METHOD M_Execute
//////////////////
//  Method Calls 
/////////////////

VAR 
	// Method local variables (reinitialized at each cycle) 

END_VAR
IF NOT bInit THEN
	M_Init();
END_IF


SUPER^.M_Execute() ;
END_METHOD

METHOD M_Init
VAR_INPUT
END_VAR

VAR

END_VAR
ParamPnom := 2200.0 ;
IN_SetptPlimit_Local :=  2200.0;
ParamQnom := 1650;
bInit := TRUE;
END_METHOD

{attribute 'object_name' := 'M_Read'}
METHOD M_Read
//////////
// Read Method for SMA : Modbus reading
//////////
VAR
	// Method local variables (reinitialized at each cycle) 
	MW 					: FB_MergeWordsToDint; 
	
	
	KK					: BYTE;						 // Index to loop over modbus blocks. 	
	JJ					: BYTE;						// Index loop over Number of SB
	CalOpTm: INT;
	
	AX_Qty				: ARRAY[1..2] OF WORD := [100, 		6 		];
	AX_Addr				: ARRAY[1..2] OF WORD := [57, 	40112 	];
	AX_UnitId			: ARRAY[1..2] OF BYTE := [1, 		1		];

	
	mesH: REAL;
	test: LREAL;
	test1: UINT;
END_VAR

IF MesDataExd.MesData.MesCP_Read THEN 
	
	FOR KK := 1 TO 1 DO
		ModbusReadRegs[KK]
		(
			nTcpPort := ParamTcpPort,
			pDestAddr := ADR(MesBlock_Temp[KK]),
			cbLength := SIZEOF(MesBlock_Temp[KK]),
			sIPAddr := ParamIPAddress,
			tTimeout := ParamTimeout,
			nQuantity := AX_Qty[KK],
			nMBAddr := AX_Addr[KK],
			nUnitID := AX_UnitID[KK],
			ClockRead := ClockRead,
			ErrorId => ModbusAlarmsID[KK],
			ModbusReadAlarm => ModbusAlarm[KK]
		);
	END_FOR
	
	MW(WORD_STRONG := MesBlock_Temp[1][1 ] 										, SIZE :=  1, FIX :=  1, SIGNED := TRUE, 	SmaDevice := TRUE, VAR_OUT := MesDataExd.MesData.MesSetptP);
	MW(WORD_STRONG := MesBlock_Temp[1][2 ] 										, SIZE :=  1, FIX :=  1, SIGNED := TRUE, 	SmaDevice := TRUE, VAR_OUT := MesDataExd.MesData.MesP);
	MW(WORD_STRONG := MesBlock_Temp[1][4 ] 										, SIZE :=  1, FIX :=  1, SIGNED := TRUE, 	SmaDevice := TRUE, VAR_OUT := MesDataExd.MesData.MesSetptQ);
	MW(WORD_STRONG := MesBlock_Temp[1][5 ] 										, SIZE :=  1, FIX :=  1, SIGNED := TRUE, 	SmaDevice := TRUE, VAR_OUT := MesDataExd.MesData.MesQ);
	MW(WORD_STRONG := MesBlock_Temp[1][10] 										, SIZE :=  1, FIX :=  1, SIGNED := TRUE, 	SmaDevice := TRUE, VAR_OUT := MesDataExd.MesData.MesNbInvAvail);
	MW(WORD_STRONG := MesBlock_Temp[1][16] 										, SIZE :=  1, FIX :=  0, SIGNED := FALSE, 	SmaDevice := TRUE, VAR_OUT := MesDataExd.MesData.MesPState);
	MW(WORD_STRONG := MesBlock_Temp[1][18] 										, SIZE :=  1, FIX :=  0, SIGNED := FALSE, 	SmaDevice := TRUE, VAR_OUT := MesDataExd.MesData.MesQState);
	MW(WORD_STRONG := MesBlock_Temp[1][20] 										, SIZE :=  1, FIX :=  0, SIGNED := FALSE, 	SmaDevice := TRUE, VAR_OUT := MesDataExd.MesData.MesGeneState);
	MW(WORD_STRONG := MesBlock_Temp[1][30], WORD_WEAK := MesBlock_Temp[1][31]	, SIZE :=  2, FIX :=  0, SIGNED := TRUE, 	SmaDevice := TRUE, VAR_OUT := MesDataExd.MesData.MesPNomControlled);
	MW(WORD_STRONG := MesBlock_Temp[1][32], WORD_WEAK := MesBlock_Temp[1][33]	, SIZE :=  2, FIX :=  0, SIGNED := TRUE, 	SmaDevice := TRUE, VAR_OUT := MesDataExd.MesData.MesPControlled);
	MW(WORD_STRONG := MesBlock_Temp[1][34], WORD_WEAK := MesBlock_Temp[1][35]	, SIZE :=  2, FIX :=  0, SIGNED := TRUE, 	SmaDevice := TRUE, VAR_OUT := MesDataExd.MesData.MesQControlled);
	MW(WORD_STRONG := MesBlock_Temp[1][40], WORD_WEAK := MesBlock_Temp[1][41]	, SIZE :=  2, FIX :=  0, SIGNED := TRUE, 	SmaDevice := TRUE, VAR_OUT := MesDataExd.MesData.MesQNomControlled);
	MW(WORD_STRONG := MesBlock_Temp[1][42] 										, SIZE :=  1, FIX :=  0, SIGNED := FALSE, 	SmaDevice := TRUE, VAR_OUT := MesDataExd.MesData.MesWatchdog);

	
END_IF
END_METHOD

METHOD M_StartStop
//////////////////
// Start and Stop AMG
/////////////////
VAR 
	// Method local variables (reinitialized at each cycle) 

END_VAR
// Set SetptLimit to zero if Stop command
SUPER^.M_StartStop() ; 
//RS_StartStop(SET:=CmdStart,Reset1:=CmdStop); IN BASE
END_METHOD

METHOD M_StateManager
//////////////////
// Detect which is the state of the inverter. IF loss of communication MesState =0 , the last inverter state is kept .  
/////////////////

VAR 
	// Method local variables (reinitialized at each cycle) 

	
	MesGeneState: WORD;

END_VAR
MesState 			:= 0  ; 

MesGeneState:= REAL_TO_WORD(MesDataExd.MesGeneState);


IF MesGeneState.0 THEN
	MesState.5 := TRUE;
ELSIF MesGeneState.1 THEN
	MesState.5 := FALSE;
END_IF

IF MesGeneState.8 = 1 THEN
	MesState.3 := TRUE;
ELSIF MesGeneState.9 THEN
	MesState.3 := FALSE;
END_IF

IF MesDataExd.MesPState = 2 THEN 
	MesState.1 := TRUE;
ELSE 
	MesState.1 := FALSE;
END_IF
IF MesDataExd.MesQState = 2 THEN 
	MesState.2 := TRUE;
ELSE 
	MesState.2 := FALSE;
END_IF
SUPER^.M_StateManager() ;
END_METHOD

{attribute 'object_name' := 'M_Write'}
METHOD M_Write
//////////////////
// Write Curtail Command through modbus to PV inverters.  
//////////////////
VAR 
	// Method local variables (reinitialized at each cycle) 

	SFW : FB_SplitRealToWords_IEEE754;

	dwordTest: DWORD;
	wordTest1: WORD;
	WordTest2: WORD;
END_VAR


AX_CmdWrite[1] := 0;
SFW(IN_Real := A1_SUBMV.A1_GRID.MesDataExd.MesData.OUT_SetptP , 	OUT_WordStrong =>AX_CmdWrite[3], 	OUT_WordWeak =>AX_CmdWrite[2]);

AX_CmdWrite[14] := 0;
SFW(IN_Real := A1_SUBMV.A1_GRID.MesDataExd.MesData.OUT_SetptQ, 	OUT_WordStrong =>AX_CmdWrite[16], 	OUT_WordWeak =>AX_CmdWrite[15]);

(*
AX_CmdWrite[31] := REAL_TO_WORD(RtuData.SetptQfU_Acknw*100);
AX_CmdWrite[37] := UINT_TO_WORD(REAL_TO_UINT(RtuData.SetptPF_Acknw*10000));
AX_CmdWrite[49] := REAL_TO_WORD(2.0); 								// Configuration of active power control (Active power control with P(f) generic 2-5)
AX_CmdWrite[50] := UINT_TO_WORD(RtuData.OUT_TypeConsigneReactive); //Type de consigne  en cours 0: Aucune, 1: Q, 2: QfU, 3: PF

*)
//
//
SFW(IN_Real := A1_SUBMV.MesDataExd.MesData.MesPsol, 			OUT_WordStrong =>AX_CmdWrite1[2], 	OUT_WordWeak =>AX_CmdWrite1[1]);


SFW(IN_Real := A1_SUBMV.MesDataExd.MesData.MesQsol, 			OUT_WordStrong =>AX_CmdWrite1[4], 	OUT_WordWeak =>AX_CmdWrite1[3]);
AX_CmdWrite1[5] := REAL_TO_WORD(REAL_TO_UINT(A1_SUBMV.MesDataExd.MesData.MesU*100));
AX_CmdWrite1[6] := REAL_TO_WORD(REAL_TO_UINT(A1_SUBMV.MesDataExd.MesData.MesFreq*100)); 
//AX_CmdWrite1[7] := REAL_TO_WORD(REAL_TO_UINT(A1_SUBMV.MesDataExd.MesData.MesTanPhi*1000)); 	// Csophi 

ModbusWrite[1]
(
	pSrcAddr := ADR(AX_CmdWrite),
	sIPAddr := ParamIPAddress,
	nTCPport := ParamTcpPort,
	tTimeout := ParamTimeout,
	nMBAddr := 133,
	cbLength := SIZEOF(AX_CmdWrite),
	nQuantity :=  50,
	WriteCmd := ClockWrite,
	nUnitID := 1
);

ModbusWrite[2]
(
	pSrcAddr := ADR(AX_CmdWrite1),
	sIPAddr := ParamIPAddress,
	nTCPport := ParamTcpPort,
	tTimeout := ParamTimeout,
	nMBAddr := 189,
	cbLength := SIZEOF(AX_CmdWrite1),
	nQuantity :=  7,
	WriteCmd := ClockWrite,
	nUnitID := 1
);

SUPER^.M_Write() ;
END_METHOD

END_FUNCTION_BLOCK

// ---- 01_Equipement_Library/ProtectRelay/FB_ProtectRelay_DM2.TcPOU
FUNCTION_BLOCK FB_ProtectRelay_DM2 EXTENDS FB_ProtectRelay_Base
//////////////////
// REF615 + REU615 : communication not allowed by EDF 

VAR_OUTPUT
	//Child objects

END_VAR

VAR_INPUT
	IN_AlarmIMax_IO								: BOOL; //Max I Alarm, Losing autorisation and not possible to consumed
	IN_AlarmUmin_IO									: BOOL; //Min U , Keeping autorisation, If we have 3 gte in 30 min ==> Stop fedding and consumed during 2h
	IN_MesWatchdogREU615_IO						: BOOL:=TRUE ;// Watchdog . 0= alarm
	MesDataExd		: ProtectRelay_Standard ; 	
END_VAR

VAR
	//M_ALARMMANAGEMENT VARIABLES//

	
	// EVALUATE //
	TON_GteIsLong	: TON ; 
	
	


		
END_VAR

METHOD M_AlarmManagement
//////////////////
// Manages Sepam Alarms. Alarms opens HT CB until Sepam manual Reset . Warning Opens CB-L but does not maintain warning
/////////////////

VAR 
	// Method local variables (reinitialized at each cycle) 
	FB_AlarmCodeManager 	: FB_AlarmCodeManager ; 

 
END_VAR


// ALARM CODE //
	FB_AlarmCodeManager(
		bAlarm1				:= MesDataExd.MesData.MesAlarmImax , 						// Max I>>0  fault 	 	
		bAlarm2				:= MesDataExd.MesData.MesAlarmUmin ,							// GTE fault 
		bAlarm3				:= MesDataExd.MesData.MesAlarmCom,						// Communication Alarm #COM
		bAlarm4				:= NOT IN_MesWatchDog_IO, 						// Watchdog REF615 not received      #COM 
		bAlarm5				:= NOT IN_MesWatchdogREU615_IO, 				// Watchdog REU615 not received	 #COM
		bAlarm6				:= FALSE, 									// 
		bAlarm7				:= FALSE, 									//
		bAlarm8				:= FALSE,                                   //
		bAlarm9				:= FALSE,                                   //
		bAlarm10			:= FALSE,                                   //
		bAlarm11			:= FALSE,                                   //
		bAlarm12			:= FALSE,                                   //
		bAlarm13			:= FALSE, 									//
		bAlarm14			:= FALSE, 									//
		bAlarm15			:= FALSE ,									// 
		wAlarmCode			=>MesDataExd.MesData.MesAlarmCode);

// WARNING CODE //
	FB_AlarmCodeManager(
		bAlarm1			:= FALSE , //
		bAlarm2			:= FALSE , //	
		bAlarm4			:= MesDataExd.MesData.MesAlarmUmin_Long, 						// GTE long 
		bAlarm5			:= FALSE, 									//
		bAlarm6			:= FALSE,                                   //
		bAlarm7			:= FALSE,                                   //
		bAlarm8			:= FALSE,                                   //
		bAlarm9			:= FALSE,                                   //
		bAlarm10		:= FALSE,                                   //
		bAlarm11		:= FALSE,                                   //
		bAlarm12		:= FALSE,                                   //
		bAlarm13		:= FALSE,                                   //
		bAlarm14		:= FALSE,                                   //
		bAlarm15		:= FALSE, 									//
		wAlarmCode		=>MesDataExd.MesData.MesWarningCode);

// EVENT CODE //
	FB_AlarmCodeManager(
		bAlarm1			:=FALSE, 		//  
		bAlarm2			:=FALSE, 		//  
		bAlarm3			:=FALSE, 		//  
		bAlarm4			:=FALSE, 		// 
		bAlarm5			:=FALSE,        //
		bAlarm6			:=FALSE,        //
		bAlarm7			:=FALSE,        //
		bAlarm8			:=FALSE,        //
		bAlarm9			:=FALSE,        //
		bAlarm10		:=FALSE,        //
		bAlarm11		:=FALSE,        //
		bAlarm12		:=FALSE,        //
		bAlarm13		:=FALSE,        //
		bAlarm14		:=FALSE,        //
		bAlarm15		:=FALSE, 
		wAlarmCode		=>MesDataExd.MesData.MesEventCode);
END_METHOD

METHOD M_CP
//////////////////
//  Emulator
/////////////////

VAR 
	// Method local variables (reinitialized at each cycle) 
	
END_VAR


SUPER^.M_CP() ; 




Trig_Cmd_Read(CLK:=IN_CmdToggleRead);
Trig_Cmd_Write(CLK:=IN_CmdToggleWrite);
	
IF Trig_Cmd_Read.Q THEN
	IN_CmdToggleRead := FALSE;
	MesDataExd.MesData.MesCP_Read := NOT MesDataExd.MesData.MesCP_Read;
END_IF


IF Trig_Cmd_Write.Q THEN
	IN_CmdToggleWrite := FALSE;
	MesDataExd.MesData.MesCP_Write := NOT MesDataExd.MesData.MesCP_Write;
END_IF
END_METHOD

METHOD M_Evaluate
VAR_INPUT
END_VAR
//Need to check the GTE FAULT


// GTE IS LONG AFTER 50S
TON_GteIsLong(IN:=IN_AlarmUmin_IO ,PT:=T#50S); 
MesDataExd.MesData.MesAlarmUmin_Long := TON_GteIsLong.Q ; 


//Update MesData

MesDataExd.MesData.MesAlarmUmin 			:= IN_AlarmUmin_IO;

TON_ComAlarm(IN:=NOT IN_MesWatchDog_IO OR NOT IN_MesWatchdogREU615_IO , PT:=ParamTempoComAlarm ) ; 
MesDataExd.MesData.MesAlarmCom		:=TON_ComAlarm.Q  ; 
MesDataExd.MesData.MesAlarmImax		:= IN_AlarmIMax_IO;
END_METHOD

END_FUNCTION_BLOCK

// ---- 01_Equipement_Library/ProtectRelay/FB_ProtectRelay_Base.TcPOU
FUNCTION_BLOCK FB_ProtectRelay_Base
//////////////////
// SEPAM system for High Voltage or Low Voltage Grid Protection. 
//////////////////
VAR_INPUT PERSISTENT
	// Parameters of the Object (instance/model specific) 
		ParamTempoComAlarm					: TIME := T#10S;	(* (s) Config : Tempo to detect LOC Alarm*)
		ParamTimeOut						: TIME := T#5S;		(* (s) Modbus Timeout*)
		ParamClockReadTime					: TIME := T#2S;		(* (s) Modbus Read Frequency*)
		ParamClockWriteTime					: TIME := T#1S;		(* (s) Modbus Write Frequency*)
				   		                    		
END_VAR                                                        

VAR_OUTPUT
	//Child objects
	
END_VAR

VAR_INPUT
	IN_CmdReset_L							: BOOL;				// (NA) External Reset Command	
    IN_CmdToggleRead						: BOOL;
    IN_CmdToggleWrite						: BOOL;
	                                    
	// I/O Inputs                       
		// GTE Protection LV            
		// WatchDog                     
	IN_MesWatchDog_IO						: BOOL :=TRUE;		// Watchdog is at True := Sepam OK
END_VAR

VAR
	//M_ALARMMANAGEMENT VARIABLES//                                                  
		TON_ComAlarm						: TON ; 			// Tempo before detecting loss of communication. 
	
	//M_READ //
		TP1									: TP;
		TP2									: TP;
		ClockRead				AT %Q*		: BOOL;
		ClockWrite							: BOOL;
	///MesDataExd						: ProtectRelay;		

    //M_CP VARIABLES//
		Trig_Cmd_Read						: R_TRIG;                                                                                        
		Trig_Cmd_Write						: R_TRIG;                                                                                        
	//M_INIT VARIABLES // 	        		
		bInit								: BOOL := TRUE ; 		// (NA) Initialize object parameters at first cycle 
END_VAR

METHOD M_AlarmManagement
//////////////////
// Manages Sepam Alarms. Alarms opens HT CB until Sepam manual Reset . Warning Opens CB-L but does not maintain warning
/////////////////

VAR 
	// Method local variables (reinitialized at each cycle) 
	FB_AlarmCodeManager 	: FB_AlarmCodeManager ; 

 
END_VAR
END_METHOD

METHOD M_CP 
VAR_INPUT
END_VAR
END_METHOD

METHOD M_Evaluate
VAR_INPUT
END_VAR
END_METHOD

METHOD M_Execute
//////////////////
//  Method Calls 
/////////////////

VAR 
	// Method local variables (reinitialized at each cycle) 

END_VAR
	TP1(IN:=NOT TP1.Q , PT:= ParamClockReadTime);
	ClockRead 		:= TP1.Q;
	TP2(IN:=NOT TP2.Q , PT:= ParamClockWriteTime);
	ClockWrite		:= TP2.Q;

// INITIALIZE // 
	IF bInit THEN
		M_Init() ; 
		bInit		:= FALSE ; 
		
	ELSIF CmdInit_G OR IN_CmdReset_L THEN 
		bInit		:= TRUE ;
		
	END_IF

// METHODS CALLS // 
	M_CP();
	M_Read(); 
	
	M_Evaluate(); 
	M_Write();
	
	M_AlarmManagement();
END_METHOD

METHOD M_Init
VAR_INPUT
END_VAR
END_METHOD

METHOD M_Read
//////////////////
//  Method Calls 
/////////////////

VAR 
	// Method local variables (reinitialized at each cycle) 

END_VAR
END_METHOD

METHOD M_Write 
VAR_INPUT
END_VAR
END_METHOD

END_FUNCTION_BLOCK

// ---- 01_Equipement_Library/ProtectRelay/FB_ProtectRelay_Flair23DM.TcPOU
FUNCTION_BLOCK FB_ProtectRelay_Flair23DM EXTENDS FB_ProtectRelay_Base
//////////////////
// SEPAM system for High Voltage or Low Voltage Grid Protection. 
//////////////////
VAR_INPUT PERSISTENT
	ParamTcpPort				: UINT:=502;                       (* (NA) Tcp port *)
	ParamIPAddress				: STRING; 						   (* (NA) IP address*)
	ParamUnitID					: BYTE; 						   (* (NA) Unit ID*)
END_VAR

VAR_INPUT 
	MesDataExd	AT %Q*	: ProtectRelay_Flair23DM;     		//  MesDataExd.MesData.xd
	
END_VAR

VAR_OUTPUT
	
END_VAR

VAR_INPUT

END_VAR

VAR

	FB_ModbusRead	          	: ARRAY[1..3] OF FB_ModbusRead; 	// Modbus Read
									
	CalCP_Read					: BOOL;								
	CalCP_Write					: BOOL;
	
	MesBlock1_Temp 				: ARRAY [1..1] OF WORD ; 
	MesBlock2_Temp 				: ARRAY [1..15] OF WORD; 
	MesBlock3_Temp 				: ARRAY [1..2] OF WORD ; 
	
	AX_ModbusReadAlarm			: ARRAY[1..3] OF BOOL  ;
	AX_ModbusReadAlarmId		: ARRAY[1..3] OF UDINT ;	
END_VAR

METHOD M_AlarmManagement
//////////////////
// Manages Sepam Alarms. Alarms opens HT CB until Sepam manual Reset. Warning Opens CB-L but does not maintain warning.
/////////////////

VAR 
	// Method local variables (reinitialized at each cycle) 
	FB_AlarmCodeManager 	: FB_AlarmCodeManager ; 
 	ComWarning				: BOOL;
	ComAlarms				: BOOL;
END_VAR
// ALARM CODE //
	FB_AlarmCodeManager(
		bAlarm1			:= NOT MesDataExd.MesData.MesAlarmCom,	// Com error: the device did not respond successfully to most recent read/write request
		bAlarm2			:= FALSE,						//				
		bAlarm3			:= FALSE,   					//
		bAlarm4			:= FALSE,   					//
		bAlarm5			:= FALSE,   					//
		bAlarm6			:= FALSE, 						//
		bAlarm7			:= FALSE,   					//
		bAlarm8			:= FALSE,   					//
		bAlarm9			:= FALSE,   					//
		bAlarm10		:= FALSE,   					//
		bAlarm11		:= FALSE,   					//
		bAlarm12		:= FALSE,   					//
		bAlarm13		:= FALSE,   					//
		bAlarm14		:= FALSE,   					//
		bAlarm15		:= FALSE, 						//
		wAlarmCode		=>MesDataExd.MesData.MesAlarmCode);   	//

// WARNING CODE //
	FB_AlarmCodeManager(
		bAlarm1			:= FALSE,						//
		bAlarm2			:= FALSE,   					//
		bAlarm4			:= FALSE,   					//
		bAlarm5			:= FALSE,   					//
		bAlarm6			:= FALSE, 						//
		bAlarm7			:= FALSE,   					// 
		bAlarm8			:= FALSE,   					// 
		bAlarm9			:= FALSE,   					// 
		bAlarm10		:= FALSE,   					// 
		bAlarm11		:= FALSE,   					// 
		bAlarm12		:= FALSE,   					// 
		bAlarm13		:= FALSE,   					// 
		bAlarm14		:= FALSE,   					// 
		bAlarm15		:= FALSE, 						// 
		wAlarmCode		=>MesDataExd.MesData.MesWarningCode);	    //

// EVENT CODE //
	FB_AlarmCodeManager(
		bAlarm1			:=FALSE,						// 		
		bAlarm2			:=FALSE,   						// 		
		bAlarm3			:=FALSE,   						// 		
		bAlarm4			:=FALSE,   						// 		
		bAlarm5			:=FALSE, 						// 
		bAlarm6			:=FALSE,   						// 
		bAlarm7			:=FALSE,   						// 
		bAlarm8			:=FALSE,   						// 
		bAlarm9			:=FALSE,   						// 
		bAlarm10		:=FALSE,   						// 
		bAlarm11		:=FALSE,   						// 
		bAlarm12		:=FALSE,   						// 
		bAlarm13		:=FALSE,   						// 
		bAlarm14		:=FALSE, 						// 
		bAlarm15		:=FALSE, 						//		
		wAlarmCode		=>MesDataExd.MesData.MesEventCode); 		//
END_METHOD

METHOD M_CP
//////////////////
//  Emulator
/////////////////

VAR 
	// Method local variables (reinitialized at each cycle) 
	
END_VAR


SUPER^.M_CP() ; 




Trig_Cmd_Read(CLK:=IN_CmdToggleRead);
Trig_Cmd_Write(CLK:=IN_CmdToggleWrite);
	
IF Trig_Cmd_Read.Q THEN
	IN_CmdToggleRead := FALSE;
	MesDataExd.MesData.MesCP_Read := NOT MesDataExd.MesData.MesCP_Read;
END_IF


IF Trig_Cmd_Write.Q THEN
	IN_CmdToggleWrite := FALSE;
	MesDataExd.MesData.MesCP_Write := NOT MesDataExd.MesData.MesCP_Write;
END_IF
END_METHOD

METHOD M_Evaluate
VAR_INPUT
END_VAR

VAR
END_VAR

SUPER^.M_Evaluate() ;
END_METHOD

METHOD M_Execute
//////////////////
//  Method Calls 
/////////////////

VAR 
	// Method local variables (reinitialized at each cycle) 

END_VAR
IF NOT bInit THEN
	M_Init();
END_IF


SUPER^.M_Execute() ;
END_METHOD

METHOD M_Init
VAR_INPUT
END_VAR
binit := true;
END_METHOD

METHOD M_Read
//////////////////
//  Method Calls 
/////////////////

VAR_INPUT
	
END_VAR
VAR 
	MW					: FB_MergeWordsToFloat;
END_VAR

// CP-Read / Write 



// System BMS 
IF MesDataExd.MesData.MesCP_Read  THEN	

	
	FB_ModbusRead[1]
		(
			nTCPPort		:= ParamTcpPort,
			ClockRead		:= MesDataExd.MesData.MesCP_Read AND ClockRead, 
			Reset			:= CmdClearFault_G OR IN_CmdReset_L,
			sIPAddr			:= ParamIPAddress,
			nUnitID			:= ParamUnitID, 
			tTimeout		:= T#5S,
			nQuantity		:= 1, 
			nMBAddr			:= 41000 , 
			cbLength		:= SIZEOF(MesBlock1_Temp), 
			pDestAddr		:= ADR(MesBlock1_Temp) , 
			ModbusReadAlarm	=> AX_ModbusReadAlarm[1] , 
			ErrorId			=> AX_ModbusReadAlarmId[1]
		);
		
	FB_ModbusRead[2]
		(
			nTCPPort		:= ParamTcpPort,
			ClockRead		:= MesDataExd.MesData.MesCP_Read AND ClockRead, 
			Reset			:= CmdClearFault_G OR IN_CmdReset_L,
			sIPAddr			:= ParamIPAddress,
			nUnitID			:= ParamUnitID, 
			tTimeout		:= T#5S,
			nQuantity		:= 14, 
			nMBAddr			:= 41200, 
			cbLength		:= SIZEOF(MesBlock2_Temp), 
			pDestAddr		:= ADR(MesBlock2_Temp) , 
			ModbusReadAlarm	=> AX_ModbusReadAlarm[2], 
			ErrorId			=> AX_ModbusReadAlarmId[2]
		);
	
	FB_ModbusRead[3]
		(
			nTCPPort		:= ParamTcpPort,
			ClockRead		:= MesDataExd.MesData.MesCP_Read AND ClockRead, 
			Reset			:= CmdClearFault_G OR IN_CmdReset_L,
			sIPAddr			:= ParamIPAddress ,
			nUnitID			:= ParamUnitID, 
			tTimeout		:= T#5S,
			nQuantity		:= 2, 
			nMBAddr			:= 41350 , 
			cbLength		:= SIZEOF(MesBlock3_Temp), 
			pDestAddr		:= ADR(MesBlock3_Temp) , 
			ModbusReadAlarm	=> AX_ModbusReadAlarm[3], 
			ErrorId			=> AX_ModbusReadAlarmId[3]
		);
			
	//COM
	MesDataExd.MesStateCom 			:= WORD_TO_BOOL(MesBlock1_Temp[1]);
	//I
	MesDataExd.MesData.MesI1 		:= WORD_TO_INT(Mesblock2_Temp[1]) ;
	MesDataExd.MesData.MesI2 	    := WORD_TO_INT(Mesblock2_Temp[2]) ;
	MesDataExd.MesData.MesI3       := WORD_TO_INT(Mesblock2_Temp[3]) ;
	MesDataExd.MesData.MesI0 	    := WORD_TO_INT(Mesblock2_Temp[4]) ;
	//Imax
	MesDataExd.MesData.MesImax1 	:= WORD_TO_INT(Mesblock2_Temp[5]) ;	
	MesDataExd.MesData.MesImax2 	:= WORD_TO_INT(Mesblock2_Temp[6]) ;	
	MesDataExd.MesData.MesImax3 	:= WORD_TO_INT(Mesblock2_Temp[7]) ;	
	//V
	MesDataExd.MesV1				:= WORD_TO_REAL(Mesblock2_Temp[8]) * 0.01 ;	
	MesDataExd.MesV2				:= WORD_TO_REAL(Mesblock2_Temp[9]) * 0.01 ;
	MesDataExd.MesV3				:= WORD_TO_REAL(Mesblock2_Temp[10])* 0.01 ;
	MesDataExd.MesV0				:= WORD_TO_REAL(Mesblock2_Temp[11])* 0.01 ;
		
	MesDataExd.MesData.MesU12		:= WORD_TO_REAL(Mesblock2_Temp[12])* 0.01 ;					// U21 
	MesDataExd.MesData.MesU23		:= WORD_TO_REAL(Mesblock2_Temp[13])* 0.01 ; 				// U32 
	MesDataExd.MesData.MesU31		:= WORD_TO_REAL(Mesblock2_Temp[14])* 0.01 ; 				// U31  
		
	MesDataExd.ControlWord 			:= MesBlock3_Temp[1];
	MesDataExd.StatusWord 			:= MesBlock3_Temp[2];
		
END_IF
END_METHOD

END_FUNCTION_BLOCK

// ---- 01_Equipement_Library/ProtectRelay/FB_ProtectRelay_MaxI.TcPOU
FUNCTION_BLOCK FB_ProtectRelay_MaxI EXTENDS FB_ProtectRelay_Base
//////////////////
// SEPAM system for High Voltage or Low Voltage Grid Protection . 
//////////////////


VAR_INPUT PERSISTENT 
	ParamTcpPort				: UINT:=502;	(* TCP Port parameter*)
	ParamIPAddress				: STRING; 		(* IP Address*)
	ParamUnitID					: BYTE; 		(* Unit ID*)
	
END_VAR

VAR_INPUT
	MesDataExd					: ProtectRelay_Standard;
END_VAR

VAR
	ClockReadInput				: BOOL;
	AX_MbRead					: ARRAY[1..1] OF FB_ModbusRead;
	AX_Word						: ARRAY[1..1] OF ARRAY[1..120] OF WORD;
	AX_ADDR						: ARRAY[1..1] OF UINT := [300];
	AX_QTY						: ARRAY[1..1] OF UINT := [16];	
	AX_UnId						: ARRAY[1..1] OF BYTE := [3];
END_VAR

METHOD M_AlarmManagement
//////////////////
// Manages Sepam Alarms. Alarms opens HT CB until Sepam manual Reset . Warning Opens CB-L but does not maintain warning
/////////////////

VAR 
	// Method local variables (reinitialized at each cycle) 
	FB_AlarmCodeManager 	: FB_AlarmCodeManager ; 
	RS_Trip					: SR;
END_VAR

MesDataExd.MesData.MesComAlarm		:= AX_MbRead[1].ModbusReadAlarm  ;

// ALARM CODE //
	FB_AlarmCodeManager(
		bAlarm1				:= MesDataExd.MesData.MesComAlarm,		// Communication alarm
		bAlarm2				:= FALSE,
		bAlarm3				:= FALSE,
		bAlarm4				:= FALSE,
		bAlarm5				:= FALSE,         					
		bAlarm6				:= FALSE, 							
		bAlarm7				:= FALSE, 
		bAlarm8				:= FALSE, 
		bAlarm9				:= FALSE, 
		bAlarm10			:= FALSE, 
		bAlarm11			:= FALSE, 
		bAlarm12			:= FALSE, 
		bAlarm13			:= FALSE, 
		bAlarm14			:= FALSE, 
		bAlarm15			:= FALSE , 	
		wAlarmCode			=> MesDataExd.MesData.MesAlarmCode);
END_METHOD

METHOD M_CP
//////////////////
//  Emulator
/////////////////

VAR 
	// Method local variables (reinitialized at each cycle) 
	
END_VAR


SUPER^.M_CP() ; 




Trig_Cmd_Read(CLK:=IN_CmdToggleRead);
Trig_Cmd_Write(CLK:=IN_CmdToggleWrite);
	
IF Trig_Cmd_Read.Q THEN
	IN_CmdToggleRead := FALSE;
	MesDataExd.MesData.MesCP_Read := NOT MesDataExd.MesData.MesCP_Read;
END_IF


IF Trig_Cmd_Write.Q THEN
	IN_CmdToggleWrite := FALSE;
	MesDataExd.MesData.MesCP_Write := NOT MesDataExd.MesData.MesCP_Write;
END_IF
END_METHOD

METHOD M_Evaluate
VAR_INPUT
END_VAR

VAR
END_VAR
END_METHOD

METHOD M_Init
VAR_INPUT
END_VAR
END_METHOD

METHOD M_Read
//////////////////
//  Method Calls 
/////////////////

VAR_INPUT
	
END_VAR
VAR 
	MW					: FB_MergeWordsToFloat;
	


	KK: INT;
END_VAR
IF MesDataExd.MesData.MesCP_Read THEN

	FOR KK := 1 TO 1 DO
		AX_MbRead[KK]
		(
			pDestAddr := ADR(AX_Word[KK]),
			sIPAddr := ParamIPAddress,
			tTimeout := T#2S,
			nTcpPort := ParamTcpPort,
			nQuantity := AX_QTY[KK],
			nMBAddr := AX_ADDR[KK],
			cbLength := SIZEOF(AX_Word[KK]),
			nUnitID := AX_UnId[KK],
			ClockRead := ClockRead
		);
	END_FOR
	
	MW(WORD_STRONG_F := AX_WORD[1][1], WORD_WEAK_F := AX_Word[1][2], NUMBER_F := MesDataExd.MesData.MesI1);
	MW(WORD_STRONG_F := AX_WORD[1][3], WORD_WEAK_F := AX_Word[1][4], NUMBER_F := MesDataExd.MesData.MesI2);
	MW(WORD_STRONG_F := AX_WORD[1][5], WORD_WEAK_F := AX_Word[1][6], NUMBER_F := MesDataExd.MesData.MesI3);
	MW(WORD_STRONG_F := AX_WORD[1][7], WORD_WEAK_F := AX_Word[1][8], NUMBER_F := MesDataExd.MesData.MesI0);
	
END_IF

MesDataExd.MesData.MesI := (MesDataExd.MesData.MesI1 + MesDataExd.MesData.MesI2 + MesDataExd.MesData.MesI3)/3;
END_METHOD

END_FUNCTION_BLOCK

// ---- 01_Equipement_Library/ProtectRelay/FB_ProtectRelay_Micom.TcPOU
FUNCTION_BLOCK FB_ProtectRelay_Micom EXTENDS FB_ProtectRelay_Base
//////////////////
// SEPAM system for High Voltage or Low Voltage Grid Protection. 
//////////////////

VAR_INPUT PERSISTENT
	// Parameters of the Object (instance/model specific) 
	   ParamTimeoutRTU						: TIME  := T#10S;					(* (s)	  Com RTU Timeout *)
	   ParamUnitID							: BYTE 	:= 1;						(* (NA)	  unit ID*)
	   ParamInInterfaceSub					: BOOL;								(* (NA)   Serial interface RS422/RS485 TYPE (0:EL6021, 1:SUB9)*)
END_VAR

VAR_OUTPUT
	//Child objects
	OUT_Protect_GTE_LONG_Running			: BOOL; 							// Long GTE fault, PP stop for 2m and lost of autorisation 

END_VAR

VAR_INPUT
	// I/O Inputs	
	IN_MesAlarmIMax_IO						: BOOL; 							// I max fault Fault, Losing autorisation and not possible to consumed
	IN_MesAlarmUmin_IO						: BOOL; 							// U min Fault, Keeping autorisation, If we have 3 gte in 30 min ==> Stop fedding and consumed during 2h
	IN_MesAlarmPWH_IO						: BOOL; 							// Defaut wattmétrique
	                                                								                                                	
	IN_CmdReset_3GTEFault					: BOOL; 							// 3GTE Fault Reset 
	
	IN_MesAlarm_GTE3Time_IO					: BOOL;								// C13-100 default        			
	IN_MesAlarmUmin_Long_IO	                : BOOL;                             // GTE default            
	IN_MesHomopol_Def_IO				    : BOOL;                             // Homopolar power default
	
	
	MesDataExd						 		: ProtectRelay_Micom; 	
END_VAR

VAR
	//M_Read
	Trig_Read								: R_TRIG;
	ModbusRTU								: FB_ModbusRTU ;					// (NA) FB for Modbus Reading
	MbStruct								: ARRAY[1..2] OF Struct_InputRTU;

                                			
	ModbusAlarm								: ARRAY[1..2] OF BOOL;				// (NA) Read alarm
	AX_Quantity								: ARRAY[1..2] OF WORD;				// (NA) Quantity of blocks to read
	AX_Address								: ARRAY[1..2] OF WORD;				// (NA) Start address of the read
	OutErrorMbRead							: ARRAY[1..2] OF BOOL;
                                			
	Busy									: BOOL;
	MesBlock_Temp							: ARRAY [1..2] OF ARRAY [0..94] OF WORD;
	                            			
	RTrigI									: R_TRIG;
	//MesDataExd						 		: ProtectRelay_Micom; 
	                            			
	//M_EVALUATE                			
	TON_GteIsLong							: TON;

	FB_3GTE									: FB_CountNinTimeWindow; 
	TP_MesAlarm_GTE3Time					: TP ;	
	TP_MesAlarmUmin_Long	                : TP ; 
	TP_MesHomopol_Def				    	: TP ; 
    TP_MesWatchdog			            	: TP ; 
END_VAR

METHOD M_AlarmManagement
//////////////////
// Manages Sepam Alarms. Alarms opens HT CB until Sepam manual reset. Warning opens CB-L but does not maintain warning.
/////////////////

VAR 
	// Method local variables (reinitialized at each cycle) 
	FB_AlarmCodeManager 	: FB_AlarmCodeManager ; 
 	ComWarning				: BOOL;
	ComAlarms				: BOOL;
END_VAR
ComWarning	:= OutErrorMbRead[1] OR OutErrorMbRead[2];
ComAlarms	:= OutErrorMbRead[1];

TON_ComAlarm			(IN:= ComAlarms , PT:= ParamTempoComAlarm, Q=> MesDataExd.MesData.MesAlarmCom) ;	
TP_MesAlarm_GTE3Time	( IN := NOT MesDataExd.MesData.MesAlarm_GTE3Time	  , PT := ParamTimeOut_Alarm ) ;
TP_MesAlarmUmin_Long	( IN := NOT MesDataExd.MesData.MesAlarmUmin_Long	  , PT := ParamTimeOut_Alarm ) ;
TP_MesHomopol_Def		( IN := NOT MesDataExd.MesHomopol_Def				  , PT := ParamTimeOut_Alarm ) ;
TP_MesWatchdog			( IN := NOT MesDataExd.MesData.MesWatchdog			  , PT := ParamTimeOut_Alarm ) ;


// ALARM CODE //
	FB_AlarmCodeManager(
		bAlarm1				:= MesDataExd.MesData.MesAlarmUmin , 		// Short GTE Fault  #Equipment
		bAlarm2				:= FALSE ,									//
		bAlarm3				:= MesDataExd.MesData.MesAlarm_GTE3Time	 ,	// C13-100 default        
		bAlarm4				:= MesDataExd.MesData.MesAlarmUmin_Long  ,  // GTE default            
		bAlarm5				:= MesDataExd.MesHomopol_Def			 ,  // Homopolar power default
		bAlarm6				:= MesDataExd.MesData.MesWatchdog		 ,  // Watchdog alarm              
		bAlarm7				:= FALSE, 									// 
		bAlarm8				:= FALSE, 									// 
		bAlarm9				:= FALSE, 									// 
		bAlarm10			:= FALSE, 									// 
		bAlarm11			:= FALSE, 									// 
		bAlarm12			:= FALSE, 									// 
		bAlarm13			:= FALSE, 									// 
		bAlarm14			:= FALSE, 									// 
		bAlarm15			:= FALSE ,									//  	
		wAlarmCode			=>MesDataExd.MesData.MesAlarmCode);

// WARNING CODE //
	FB_AlarmCodeManager(
		bAlarm1			:= ComWarning, 									// At least one register do not respond #COM #Equipment
		bAlarm2			:= MesDataExd.MesData.MesAlarmCom ,				// Communication alarm #COM  #Equipment
		bAlarm3			:= FALSE , 										//		
		bAlarm4			:= FALSE , 										//
		bAlarm5			:= FALSE , 										//
		bAlarm6			:= FALSE , 										//
		bAlarm7			:= FALSE , 										//
		bAlarm8			:= FALSE , 										//
		bAlarm9			:= FALSE , 										//
		bAlarm10		:= FALSE, 										//
		bAlarm11		:= FALSE, 										//
		bAlarm12		:= FALSE, 										//
		bAlarm13		:= FALSE, 										//
		bAlarm14		:= FALSE, 										//
		bAlarm15		:= FALSE, 										//
		wAlarmCode		=>MesDataExd.MesData.MesWarningCode);

// EVENT CODE //
	FB_AlarmCodeManager(
		bAlarm1			:=TP_MesAlarm_GTE3Time .Q ,						// C13-100 default  back to normal       
		bAlarm2			:=TP_MesAlarmUmin_Long .Q ,						// GTE default   back to normal          
		bAlarm3			:=TP_MesHomopol_Def	   .Q ,						// Homopolar power default back to normal
		bAlarm4			:=TP_MesWatchdog	   .Q ,     				// Watchdog alarm back to normal       
		bAlarm5			:=FALSE, 										//
		bAlarm6			:=FALSE, 										//
		bAlarm7			:=FALSE, 										//
		bAlarm8			:=FALSE, 										//
		bAlarm9			:=FALSE, 										//
		bAlarm10		:=FALSE, 										//
		bAlarm11		:=FALSE, 										//
		bAlarm12		:=FALSE, 										//
		bAlarm13		:=FALSE, 										//
		bAlarm14		:=FALSE, 										//
		bAlarm15		:=FALSE, 										//
		wAlarmCode		=>MesDataExd.MesData.MesEventCode);
IF ParamNC THEN
		MesDataExd.MesData.MesAlarm_GTE3Time	:= NOT IN_MesAlarm_GTE3Time_IO	;
        MesDataExd.MesData.MesAlarmUmin_Long    := NOT IN_MesAlarmUmin_Long_IO	;
        MesDataExd.MesHomopol_Def			    := NOT IN_MesHomopol_Def_IO	    ;
        MesDataExd.MesData.MesWatchdog		    := NOT IN_MesWatchdog_IO		;  
ELSE
		MesDataExd.MesData.MesAlarm_GTE3Time	:=  IN_MesAlarm_GTE3Time_IO	;
        MesDataExd.MesData.MesAlarmUmin_Long    :=  IN_MesAlarmUmin_Long_IO	;
        MesDataExd.MesHomopol_Def			    :=  IN_MesHomopol_Def_IO	    ;
        MesDataExd.MesData.MesWatchdog		    :=  IN_MesWatchdog_IO		;  

END_IF
END_METHOD

METHOD M_Evaluate
VAR_INPUT
END_VAR

VAR

END_VAR
// GTE IS LONG AFTER 50S
//	TON_GteIsLong(IN:=IN_MesAlarmUmin_IO ,PT:=T#50S); 
//	MesDataExd.MesData.MesAlarmUmin_Long := TON_GteIsLong.Q ; 
//	
//	
//	
//	
//	FB_3GTE(IN_bInput := IN_MesAlarmUmin_IO , IN_bReset := IN_CmdReset_3GTEFault , IN_CountMax := 3 , ParamTimeToMeasure := T#30M , OUT_FlagNinT =>MesDataExd.MesData.MesAlarm_GTE3Time ) ; 
//		
//	
//	
//	
//	//Update MesData
//	MesDataExd.MesData.MesI			:= (MesDataExd.MesData.MesI1 + MesDataExd.MesData.MesI2 + MesDataExd.MesData.MesI3) / 3 ;
//	MesDataExd.MesData.MesAlarmUmin := IN_MesAlarmUmin_IO;
//	MesDataExd.MesData.MesAlarmImax	:= IN_MesAlarmIMax_IO;
//	
//	MesDataExd.MesStopPP_UminLong 	:= OUT_Protect_GTE_LONG_Running;
END_METHOD

METHOD M_Init
VAR_INPUT
END_VAR
END_METHOD

METHOD M_Read
//////////////////
//  Method Calls 
/////////////////

VAR 
	MW 					: FB_MergeWordsToDint; 
	KK : UINT;

	AX_Addr					: ARRAY[1..2] OF UINT 	:= [16#113,		16#10B];
	AX_Qty					: ARRAY[1..2] OF UINT	:= [94,			1];
	AX_UnitId				: ARRAY[1..2] OF BYTE	:= [1,			1];
	AX_Function				: ARRAY[1..2] OF UINT	:= [3,			3];	
	AX_Priority				: ARRAY[1..2] OF UINT	:= [1,			1];
END_VAR
// CP-Read / Write 

//	MesDataExd.MesData.MesCP_Read := MesCP_Read ; 
//	
//	IF MesCP_Read  THEN	
//		
//	
//	ModbusRTU();
//	Trig_Read(Clk := CalLocalTimeStruct.wMilliseconds < 200);
//	IF Trig_Read.Q THEN
//		FOR KK := 1 TO 2 DO
//				ModbusRTU.M_AddAction_FIFO(InStruct := MbStruct[KK], InPriority := AX_Priority[KK]);
//		END_FOR
//	END_IF
//	
//	MbStruct[1].InBuffer 	:= ADR(MesBlock_Temp[1]);
//	MbStruct[1].InFunction 	:= AX_Function[1];
//	MbStruct[1].InQuantity 	:= AX_Qty[1];
//	MbStruct[1].InStartAddr := AX_Addr[1];
//	MbStruct[1].InUnitID 	:= AX_UnitId[1];
//	
//	MbStruct[2].InBuffer 	:= ADR(MesBlock_Temp[2]);
//	MbStruct[2].InFunction 	:= AX_Function[2];
//	MbStruct[2].InQuantity 	:= AX_Qty[2];
//	MbStruct[2].InStartAddr := AX_Addr[2];
//	MbStruct[2].InUnitID 	:= AX_UnitId[2];
//	
//	//MW( WORD_STRONG:= MesBlock_Temp[1][0], SIGNED:=FALSE, FIX:=1 , SIZE:=1, VAR_OUT := MesDataExd.MesData.MesI1);
//	//MW( WORD_STRONG:= MesBlock_Temp[1][1], SIGNED:=FALSE, FIX:=1 , SIZE:=1, VAR_OUT := MesDataExd.MesData.MesI2);
//	//MW( WORD_STRONG:= MesBlock_Temp[1][2], SIGNED:=FALSE, FIX:=1 , SIZE:=1, VAR_OUT := MesDataExd.MesData.MesI3);
//	//MW( WORD_STRONG:= MesBlock_Temp[1][4], SIGNED:=FALSE, FIX:=1 , SIZE:=1, VAR_OUT := MesDataExd.MesData.MesI0);
//	//MW( WORD_STRONG:= MesBlock_Temp[1][8], SIGNED:=FALSE, FIX:=1 , SIZE:=1, VAR_OUT := MesDataExd.MesData.MesImax1);
//	//MW( WORD_STRONG:= MesBlock_Temp[1][9], SIGNED:=FALSE, FIX:=1 , SIZE:=1, VAR_OUT := MesDataExd.MesData.MesImax2);
//	//MW( WORD_STRONG:= MesBlock_Temp[1][10], SIGNED:=FALSE, FIX:=1 , SIZE:=1, VAR_OUT := MesDataExd.MesData.MesImax3);
//	////MW( WORD_STRONG:= MesBlock_Temp[1][14], SIGNED:=FALSE, FIX:=0 , SIZE:=1, VAR_OUT := MesDataExd.MesV1);
//	//MW( WORD_STRONG:= MesBlock_Temp[1][15], SIGNED:=FALSE, FIX:=0 , SIZE:=1, VAR_OUT := MesDataExd.MesV2);
//	//MW( WORD_STRONG:= MesBlock_Temp[1][16], SIGNED:=FALSE, FIX:=0 , SIZE:=1, VAR_OUT := MesDataExd.MesV3);
//	//MW( WORD_STRONG:= MesBlock_Temp[1][11], SIGNED:=FALSE, FIX:=0 , SIZE:=1, VAR_OUT := MesDataExd.MesData.MesU12);
//	//MW( WORD_STRONG:= MesBlock_Temp[1][12], SIGNED:=FALSE, FIX:=0 , SIZE:=1, VAR_OUT := MesDataExd.MesData.MesU31);
//	//MW( WORD_STRONG:= MesBlock_Temp[1][13], SIGNED:=FALSE, FIX:=0 , SIZE:=1, VAR_OUT := MesDataExd.MesData.MesU23);
//	//MW( WORD_STRONG:= MesBlock_Temp[1][20], SIGNED:=FALSE, FIX:=2 , SIZE:=1, VAR_OUT := MesDataExd.MesData.MesFreq);
//	//MW( WORD_STRONG:= MesBlock_Temp[1][21], SIGNED:=TRUE, FIX:=0 , SIZE:=1, VAR_OUT := MesDataExd.MesP);
//	//MW( WORD_STRONG:= MesBlock_Temp[1][22], SIGNED:=TRUE, FIX:=0 , SIZE:=1, VAR_OUT := MesDataExd.MesQ);
//	//MW( WORD_STRONG:= MesBlock_Temp[1][23], SIGNED:=TRUE, FIX:=0 , SIZE:=1, VAR_OUT := MesDataExd.MesS);
//	//MW( WORD_STRONG:= MesBlock_Temp[1][26], SIGNED:=TRUE, FIX:=2 , SIZE:=1, VAR_OUT := MesDataExd.MesCosPhi);
//	//MW( WORD_STRONG:= MesBlock_Temp[1][27], WORD_WEAK := MesBlock_Temp[1][28], SIGNED:=FALSE, FIX:=1 , SIZE:=2, VAR_OUT := MesDataExd.EActProd);
//	//MW( WORD_STRONG:= MesBlock_Temp[1][29], WORD_WEAK := MesBlock_Temp[1][30], SIGNED:=FALSE, FIX:=1 , SIZE:=2, VAR_OUT := MesDataExd.EActCons);
//	//MW( WORD_STRONG:= MesBlock_Temp[1][31], WORD_WEAK := MesBlock_Temp[1][32], SIGNED:=FALSE, FIX:=1 , SIZE:=2, VAR_OUT := MesDataExd.EReactProd);
//	//MW( WORD_STRONG:= MesBlock_Temp[1][33], WORD_WEAK := MesBlock_Temp[1][34], SIGNED:=FALSE, FIX:=1 , SIZE:=2, VAR_OUT := MesDataExd.EReactCons);
//	
//	
//	MesDataExd.Input11 := MesBlock_Temp[2][0].0;
//	MesDataExd.Input12 := MesBlock_Temp[2][0].1;
//	MesDataExd.Input13 := MesBlock_Temp[2][0].2;
//	MesDataExd.Input14 := MesBlock_Temp[2][0].3;
//	MesDataExd.Input21 := MesBlock_Temp[2][0].4;
//	MesDataExd.Input22 := MesBlock_Temp[2][0].5;
//	MesDataExd.Input23 := MesBlock_Temp[2][0].6;
//	MesDataExd.Input24 := MesBlock_Temp[2][0].7;
//	MesDataExd.Input25 := MesBlock_Temp[2][0].8;
//	MesDataExd.Input26 := MesBlock_Temp[2][0].9;
//	
//	END_IF
//	
//	//// Properties Update 
//	//MesDataExd.MesU := (MesDataExd.MesData.MesU12 + MesDataExd.MesData.MesU31 + MesDataExd.MesData.MesU23 ) /3 ; 
//	//
//	//IF MesDataExd.MesP <> 0 THEN
//	//MesDataExd.MesTanPhi := MesDataExd.MesQ /MesDataExd.MesP;
//	//ELSE
//	//MesDataExd.MesTanPhi := 0;
//	//END_IF
END_METHOD

END_FUNCTION_BLOCK

// ---- 01_Equipement_Library/ProtectRelay/FB_ProtectRelay_NSXCB.TcPOU
FUNCTION_BLOCK FB_ProtectRelay_NSXCB EXTENDS FB_ProtectRelay_Base
//////////////////
// SEPAM system for High Voltage or Low Voltage Grid Protection. 
//////////////////
VAR_INPUT PERSISTENT
	ParamTcpPort				: UINT:=502;		(* (NA) Tcp port *)
	ParamIPAddress				: STRING;           (* (NA) IP address*)
	ParamUnitID					: BYTE;             (* (NA) Unit ID*)
END_VAR

VAR_INPUT 

END_VAR

VAR_OUTPUT
	
END_VAR

VAR_INPUT
MesDataExd	AT %Q*	: ProtectRelay_NSXCB;
END_VAR

VAR

	
	FB_ModbusRead	          	: ARRAY[1..3] OF FB_ModbusRead; 
		
	CalCP_Read					: BOOL;
	CalCP_Write                 : BOOL;
	
	MesBlock1_Temp 				: ARRAY [1..1] OF WORD ; 
	MesBlock2_Temp 				: ARRAY [1..32] OF WORD ; 
	MesBlock3_Temp 				: ARRAY [1..8] OF WORD ; 
	
	AX_ModbusReadAlarm			: ARRAY[1..3] OF BOOL;
	AX_ModbusReadAlarmId		: ARRAY[1..3] OF UDINT;	
END_VAR

METHOD M_AlarmManagement
//////////////////
// Manages Sepam Alarms. Alarms opens HT CB until Sepam manual Reset. Warning Opens CB-L but does not maintain warning.
/////////////////

VAR 
	// Method local variables (reinitialized at each cycle) 
	FB_AlarmCodeManager 	: FB_AlarmCodeManager; 
 	ComWarning				: BOOL;
	ComAlarms				: BOOL;
END_VAR

// ALARM CODE //
	FB_AlarmCodeManager(
		bAlarm1			:= NOT MesDataExd.MesData.MesAlarmCom,	//
		bAlarm2			:= FALSE,						//
		bAlarm3			:= FALSE,						//
		bAlarm4			:= FALSE,						//     							
		bAlarm5			:= FALSE,						//         						 
		bAlarm6			:= FALSE, 						// 
		bAlarm7			:= FALSE,   					//
		bAlarm8			:= FALSE,   					//
		bAlarm9			:= FALSE,   					//
		bAlarm10		:= FALSE,   					//
		bAlarm11		:= FALSE,   					//
		bAlarm12		:= FALSE,   					//
		bAlarm13		:= FALSE,   					//
		bAlarm14		:= FALSE,   					//
		bAlarm15		:= FALSE, 						// Command Alarm in case of intervention
		wAlarmCode		=>MesDataExd.MesData.MesAlarmCode);

// WARNING CODE //
	FB_AlarmCodeManager(
		bAlarm1			:= FALSE,						//
		bAlarm2			:= FALSE,   					//
		bAlarm4			:= FALSE,   					//
		bAlarm5			:= FALSE,   					//
		bAlarm6			:= FALSE,						//
		bAlarm7			:= FALSE,   					//
		bAlarm8			:= FALSE,   					//
		bAlarm9			:= FALSE,   					//
		bAlarm10		:= FALSE, 						//
		bAlarm11		:= FALSE,   					//
		bAlarm12		:= FALSE,   					//
		bAlarm13		:= FALSE,   					//
		bAlarm14		:= FALSE,   					//
		bAlarm15		:= FALSE,   					//
		wAlarmCode		=>MesDataExd.MesData.MesWarningCode);		//

// EVENT CODE //
	FB_AlarmCodeManager(
		bAlarm1			:=FALSE, 						// 
		bAlarm2			:=FALSE, 						// 
		bAlarm3			:=FALSE, 						// 
		bAlarm4			:=FALSE, 						// 
		bAlarm5			:=FALSE, 						//
		bAlarm6			:=FALSE,        				//
		bAlarm7			:=FALSE,        				//
		bAlarm8			:=FALSE,        				//
		bAlarm9			:=FALSE, 						//
		bAlarm10		:=FALSE,        				//
		bAlarm11		:=FALSE,        				//
		bAlarm12		:=FALSE,        				//
		bAlarm13		:=FALSE,        				//
		bAlarm14		:=FALSE,        				//
		bAlarm15		:=FALSE,        				//
		wAlarmCode		=>MesDataExd.MesData.MesEventCode);		//
END_METHOD

METHOD M_CP
//////////////////
//  Emulator
/////////////////

VAR 
	// Method local variables (reinitialized at each cycle) 
	
END_VAR


SUPER^.M_CP() ; 




Trig_Cmd_Read(CLK:=IN_CmdToggleRead);
Trig_Cmd_Write(CLK:=IN_CmdToggleWrite);
	
IF Trig_Cmd_Read.Q THEN
	IN_CmdToggleRead := FALSE;
	MesDataExd.MesData.MesCP_Read := NOT MesDataExd.MesData.MesCP_Read;
END_IF


IF Trig_Cmd_Write.Q THEN
	IN_CmdToggleWrite := FALSE;
	MesDataExd.MesData.MesCP_Write := NOT MesDataExd.MesData.MesCP_Write;
END_IF
END_METHOD

METHOD M_Evaluate
VAR_INPUT
	
END_VAR

VAR
	
END_VAR
END_METHOD

METHOD M_Execute
//////////////////
//  Method Calls 
/////////////////

VAR 
	// Method local variables (reinitialized at each cycle) 

END_VAR
IF NOT bInit THEN
	M_Init();
END_IF


SUPER^.M_Execute() ;
END_METHOD

METHOD M_Init
VAR_INPUT
END_VAR
END_METHOD

METHOD M_Read
//////////////////
//  Method Calls 
/////////////////

VAR_INPUT
	
END_VAR
VAR 
	MW					: FB_MergeWordsToFloat;
	MW_1				: FB_MergeWordsToDint;
END_VAR
// CP-Read / Write 



// System BMS 
IF MesDataExd.MesData.MesCP_Read  THEN	

	FB_ModbusRead[1]
		(
			nTCPPort		:= ParamTcpPort,
			ClockRead		:= MesDataExd.MesData.MesCP_Read AND ClockRead, 
			Reset			:= CmdClearFault_G OR IN_CmdReset_L,
			sIPAddr			:= ParamIPAddress,
			nUnitID			:= ParamUnitID, 
			tTimeout		:= T#5S,
			nQuantity		:= 1, 
			nMBAddr			:= 42000 , 
			cbLength		:= SIZEOF(MesBlock1_Temp), 
			pDestAddr		:= ADR(MesBlock1_Temp), 
			ModbusReadAlarm	=> AX_ModbusReadAlarm[1] , 
			ErrorId			=> AX_ModbusReadAlarmId[1]
		);
		
	FB_ModbusRead[2]
		(
			nTCPPort		:= ParamTcpPort,
			ClockRead		:= MesDataExd.MesData.MesCP_Read AND ClockRead, 
			Reset			:= CmdClearFault_G OR IN_CmdReset_L,
			sIPAddr			:= ParamIPAddress,
			nUnitID			:= ParamUnitID, 
			tTimeout		:= T#5S,
			nQuantity		:= 32, 
			nMBAddr			:= 42420, 
			cbLength		:= SIZEOF(MesBlock2_Temp), 
			pDestAddr		:= ADR(MesBlock2_Temp) , 
			ModbusReadAlarm	=> AX_ModbusReadAlarm[2], 
			ErrorId			=> AX_ModbusReadAlarmId[2]
		);
	
	FB_ModbusRead[3]
		(
			nTCPPort		:= ParamTcpPort,
			ClockRead		:= MesDataExd.MesData.MesCP_Read AND ClockRead, 
			Reset			:= CmdClearFault_G OR IN_CmdReset_L,
			sIPAddr			:= ParamIPAddress ,
			nUnitID			:= ParamUnitID, 
			tTimeout		:= T#5S,
			nQuantity		:= 8, 
			nMBAddr			:= 42556 , 
			cbLength		:= SIZEOF(MesBlock3_Temp), 
			pDestAddr		:= ADR(MesBlock3_Temp), 
			ModbusReadAlarm	=> AX_ModbusReadAlarm[3], 
			ErrorId			=> AX_ModbusReadAlarmId[3]
		);
	
	//COM
	MesDataExd.MesStatCom 	:= WORD_TO_BOOL(MesBlock1_Temp[1]);
		 
	MW( WORD_STRONG:= MesBlock2_Temp[2  ],	WORD_WEAK := MesBlock2_Temp[1  ], VAR_OUT := MesDataExd.MesData.MesFreq 	 );	
	MW( WORD_STRONG:= MesBlock2_Temp[4  ],	WORD_WEAK := MesBlock2_Temp[3  ], VAR_OUT := MesDataExd.MesMaxFreq );
//	MW( WORD_STRONG_F:= MesBlock2_Temp[6  ],	WORD_WEAK_F := MesBlock2_Temp[5  ], NUMBER_F := MesDataExd.MesData.MesFreq	 );	
	MW( WORD_STRONG:= MesBlock2_Temp[8  ],	WORD_WEAK := MesBlock2_Temp[7  ], VAR_OUT := MesDataExd.MesP2	 	 );
	MW( WORD_STRONG:= MesBlock2_Temp[10 ],	WORD_WEAK := MesBlock2_Temp[9  ], VAR_OUT := MesDataExd.MesP3	 	 );
	MW( WORD_STRONG:= MesBlock2_Temp[12 ],	WORD_WEAK := MesBlock2_Temp[11 ], VAR_OUT := MesDataExd.MesPtot	 );                      
	MW( WORD_STRONG:= MesBlock2_Temp[14 ],	WORD_WEAK := MesBlock2_Temp[13 ], VAR_OUT := MesDataExd.MesQ1	 	 );
	MW( WORD_STRONG:= MesBlock2_Temp[16 ],	WORD_WEAK := MesBlock2_Temp[15 ], VAR_OUT := MesDataExd.MesQ2	 	 );
	MW( WORD_STRONG:= MesBlock2_Temp[18 ],	WORD_WEAK := MesBlock2_Temp[17 ], VAR_OUT := MesDataExd.MesQ3	 	 );
	MW( WORD_STRONG:= MesBlock2_Temp[20 ],	WORD_WEAK := MesBlock2_Temp[19 ], VAR_OUT := MesDataExd.MesQtot	 );                
	MW( WORD_STRONG:= MesBlock2_Temp[22 ],	WORD_WEAK := MesBlock2_Temp[21 ], VAR_OUT := MesDataExd.MesS1	 	 );
	MW( WORD_STRONG:= MesBlock2_Temp[24 ],	WORD_WEAK := MesBlock2_Temp[23 ], VAR_OUT := MesDataExd.MesS2	 	 );
    MW( WORD_STRONG:= MesBlock2_Temp[26 ],	WORD_WEAK := MesBlock2_Temp[25 ], VAR_OUT := MesDataExd.MesS3	 	 );
	MW( WORD_STRONG:= MesBlock2_Temp[28 ],	WORD_WEAK := MesBlock2_Temp[27 ], VAR_OUT := MesDataExd.MesStot	 );  
	
	MW_1(WORD_STRONG := MesBlock2_Temp[29 ], 	WORD_WEAK := MesBlock2_Temp[30 ] ,SIZE := 2,SIGNED := 1 ,VAR_OUT := MesDataExd.MesEAct );
	MW_1(WORD_STRONG := MesBlock2_Temp[31 ], 	WORD_WEAK := MesBlock2_Temp[32 ] ,SIZE := 2,SIGNED := 1 ,VAR_OUT := MesDataExd.MesEReact );
	
	MW( WORD_STRONG:= MesBlock3_Temp[2  ],	WORD_WEAK := MesBlock3_Temp[1  ], VAR_OUT := MesDataExd.MesCosPhi1 );	
	MW( WORD_STRONG:= MesBlock3_Temp[4  ],	WORD_WEAK := MesBlock3_Temp[3  ], VAR_OUT := MesDataExd.MesCosPhi2 );
	MW( WORD_STRONG:= MesBlock3_Temp[6  ],	WORD_WEAK := MesBlock3_Temp[5  ], VAR_OUT := MesDataExd.MesCosPhi3 );	
	MW( WORD_STRONG:= MesBlock3_Temp[8  ],	WORD_WEAK := MesBlock3_Temp[7  ], VAR_OUT := MesDataExd.MesCosPhi	 );

	
END_IF
END_METHOD

END_FUNCTION_BLOCK

// ---- 01_Equipement_Library/ProtectRelay/FB_ProtectRelay_PACE100ST.TcPOU
FUNCTION_BLOCK FB_ProtectRelay_PACE100ST EXTENDS FB_ProtectRelay_Base
//////////////////
// SEPAM system for High Voltage or Low Voltage Grid Protection . 
//////////////////


VAR_INPUT PERSISTENT
	// Parameters of the Object (instance/model specific) 
	ParamInInterfaceSub						: BOOL := TRUE; // Serial interface RS422/RS485 TYPE (0:EL6021,1:SUB9)
END_VAR

VAR_OUTPUT

END_VAR

VAR_INPUT
	InUnitID            					: DINT;			// (NA)   ID FOR SEPAM S48 Modbus Unit ID. 	

	IN_MesAlarmI0Max_IO						: BOOL;
	IN_MesAlarmIMax_IO						: BOOL;
	
	MesDataExd				AT %Q* 	: ProtectRelay_PACE100ST ;
	
	
END_VAR

VAR

	ModbusRTU								: FB_ModbusRTU;
	MesBlock								: ARRAY[1..3] OF ARRAY[1..120] OF WORD;	
	AX_Addr									: ARRAY[1..3] OF UINT 	:= [1200,	1500,	2000];
	AX_Qty									: ARRAY[1..3] OF UINT	:= [2,		2,		3];
	AX_UnitId								: ARRAY[1..3] OF BYTE	:= [1,		1,		1];
	AX_Function								: ARRAY[1..3] OF UINT	:= [4,		4,		4];	
	AX_Priority								: ARRAY[1..3] OF UINT	:= [1,		1,		1];
	AX_bStart								: ARRAY[1..3] OF BOOL;
	AX_TrigRead								: ARRAY[1..3] OF R_trig;
	MbStruct								: ARRAY[1..3] OF Struct_InputRTU;	
	
	KK										: INT;


	//M_EVALUATE

	//ClockRead								: BOOL;

END_VAR

METHOD M_AlarmManagement
//////////////////
// Manages Sepam Alarms. Alarms opens HT CB until Sepam manual Reset . Warning Opens CB-L but does not maintain warning
/////////////////

VAR 
	// Method local variables (reinitialized at each cycle) 
	FB_AlarmCodeManager 	: FB_AlarmCodeManager ; 

END_VAR

// ALARM CODE //
	FB_AlarmCodeManager(
		bAlarm1				:= MesDataExd.CB_In_Alarm,		// CB in Alarm
		bAlarm2				:= IN_MesAlarmI0Max_IO,					// Max IO Fault
		bAlarm3				:= IN_MesAlarmIMax_IO,						// Max I Fault 
		bAlarm4				:= FALSE,						// 
		bAlarm5				:= FALSE,						//
		bAlarm6				:= FALSE, 						// 
		bAlarm7				:= FALSE, 						// 
		bAlarm8				:= FALSE, 						// 
		bAlarm9				:= FALSE, 						// 
		bAlarm10			:= FALSE, 						// 
		bAlarm11			:= FALSE, 						//
		bAlarm12			:= FALSE, 						// 
		bAlarm13			:= FALSE, 						//
		bAlarm14			:= FALSE, 						//
		bAlarm15			:= FALSE, 						// 
		wAlarmCode			=>MesDataExd.MesData.MesAlarmCode);

// WARNING CODE //
	FB_AlarmCodeManager(
		bAlarm1			:= FALSE,//
		bAlarm2			:= FALSE,//
		bAlarm4			:= FALSE,//
		bAlarm5			:= FALSE,//
		bAlarm6			:= FALSE,// 
		bAlarm7			:= FALSE,// 
		bAlarm8			:= FALSE,// 
		bAlarm9			:= FALSE,// 
		bAlarm10		:= FALSE,// 
		bAlarm11		:= FALSE,// 
		bAlarm12		:= FALSE,// 
		bAlarm13		:= FALSE,// 
		bAlarm14		:= FALSE,// 
		bAlarm15		:= FALSE,// 
		wAlarmCode		=>MesDataExd.MesData.MesWarningCode);

// EVENT CODE //
	FB_AlarmCodeManager(
		bAlarm1			:=FALSE, 		// 
		bAlarm2			:=FALSE, 		// 
		bAlarm3			:=FALSE, 		// 
		bAlarm4			:=FALSE, 		// 
		bAlarm5			:=FALSE, 		//
		bAlarm6			:=FALSE, 		//
		bAlarm7			:=FALSE, 		//
		bAlarm8			:=FALSE, 		//
		bAlarm9			:=FALSE, 		//
		bAlarm10		:=FALSE, 		//
		bAlarm11		:=FALSE, 		//
		bAlarm12		:=FALSE, 		//
		bAlarm13		:=FALSE, 		//
		bAlarm14		:=FALSE, 		//
		bAlarm15		:=FALSE, 		//
		wAlarmCode		=>MesDataExd.MesData.MesEventCode);
END_METHOD

METHOD M_CP
//////////////////
//  Emulator
/////////////////

VAR 
	// Method local variables (reinitialized at each cycle) 
	
END_VAR


SUPER^.M_CP() ; 




Trig_Cmd_Read(CLK:=IN_CmdToggleRead);
Trig_Cmd_Write(CLK:=IN_CmdToggleWrite);
	
IF Trig_Cmd_Read.Q THEN
	IN_CmdToggleRead := FALSE;
	MesDataExd.MesData.MesCP_Read := NOT MesDataExd.MesData.MesCP_Read;
END_IF


IF Trig_Cmd_Write.Q THEN
	IN_CmdToggleWrite := FALSE;
	MesDataExd.MesData.MesCP_Write := NOT MesDataExd.MesData.MesCP_Write;
END_IF
END_METHOD

METHOD M_Evaluate
VAR_INPUT
END_VAR

VAR
	CloseMainMVCB							: BOOL;
	Valtemp									: REAL;
	MesConnectAuthorization					: BOOL;

END_VAR
END_METHOD

METHOD M_Init
VAR_INPUT
END_VAR
//Modbus RTU Relay
FOR KK := 1 TO 4 DO 
	MbStruct[KK].InBuffer := ADR(MesBlock[KK]);
	MbStruct[KK].InFunction := AX_Function[KK];
	MbStruct[KK].InQuantity := AX_Qty[KK];
	MbStruct[KK].InStartAddr := AX_Addr[KK];
	MbStruct[KK].InUnitID := AX_UnitId[KK];
END_FOR
END_METHOD

METHOD M_Read
//////////////////
//  Method Calls 
/////////////////

VAR 
//local variables (reinitialized at each cycle) 
	MW 					: FB_MergeWordsToDint; 
	MW_Float			: FB_MergeWordsToFloat; 
END_VAR
// CP-Read / Write 


// System BMS 
IF MesDataExd.MesData.MesCP_Read  THEN	

	ModbusRTU();
	
	
	FOR KK := 1 TO 4 DO
		AX_TrigRead[KK](CLK  :=CalLocalTimeStruct.wSecond MOD 5 = 0);
		IF AX_TrigRead[KK].Q THEN
			ModbusRTU.M_AddAction_FIFO(InStruct := MbStruct[KK], InPriority := AX_Priority[KK]);
		END_IF
	END_FOR
	
	
	MW_Float( WORD_STRONG:= MesBlock[1][1], 	WORD_WEAK := MesBlock[1][2],  VAR_OUT:=MesDataExd.MesData.MesI1);
	MW_Float( WORD_STRONG:= MesBlock[1][3], 	WORD_WEAK := MesBlock[1][4],  VAR_OUT:=MesDataExd.MesData.MesI2);
	MW_Float( WORD_STRONG:= MesBlock[1][5], 	WORD_WEAK := MesBlock[1][6],  VAR_OUT:=MesDataExd.MesData.MesI3);
	MW_Float( WORD_STRONG:= MesBlock[1][7], 	WORD_WEAK := MesBlock[1][8],  VAR_OUT:=MesDataExd.MesData.MesI0);
	MW_Float( WORD_STRONG:= MesBlock[1][15], 	WORD_WEAK := MesBlock[1][16], VAR_OUT:=MesDataExd.Thermal_Overload);
	MW_Float( WORD_STRONG:= MesBlock[1][17], 	WORD_WEAK := MesBlock[1][18], VAR_OUT:=MesDataExd.MesData.MesFreq);
	
	
	MesDataExd.Comut 			:= WORD_TO_BOOL(MesBlock[2][7]);
	MesDataExd.CB_Close 		:= WORD_TO_BOOL(MesBlock[2][8]);
	MesDataExd.CB_In_Alarm 		:= WORD_TO_BOOL(MesBlock[2][9]);
	MesDataExd.Trip_Counter 	:= WORD_TO_INT(MesBlock[3][3]);

END_IF
END_METHOD

END_FUNCTION_BLOCK

// ---- 01_Equipement_Library/ProtectRelay/FB_ProtectRelay_REF615.TcPOU
FUNCTION_BLOCK FB_ProtectRelay_REF615 EXTENDS FB_ProtectRelay_Base
VAR_INPUT PERSISTENT
	{attribute 'OPC.UA.DA' := '1'} 
		ParamIPAddress				: STRING 	:= '192.168.20.66'; 	// (NA)Config: IP Adress of PV INverter
	{attribute 'OPC.UA.DA' := '1'} 
		ParamUnitID 				: BYTE  	:= 1; 			  		// (NA)   Modbus Unit ID. 
	{attribute 'OPC.UA.DA' := '1'} 
		ParamTCPPort				: UINT		:= 502;					// (NA) TCP port for modbus
		

//		ParamTempoComAlarm			: TIME 		:= T#2S;
//		ParamTempoComWarning		: TIME		:= T#2S;
		ParamNominalCurrent			: REAL 		:= 100 ; 				// (A) Nominal current set in the protection relay.
		
END_VAR

VAR_INPUT
		MesDataExd		AT %Q* 	: ProtectRelay_REFIO ; 
	
END_VAR

VAR
	// M_ALARMMANAGEMENT		
//		TON_ComAlarm				: TON;
//		TON_ComWarning				: TON;	
//		MesWarningCom				: BOOL;
//		MesAlarmCom					: BOOL;
	// M_READ VARIABLES//
		AX_ModbusRead		   		: ARRAY [1..3] OF FB_ModbusRead ; 					// (NA) FB for Modbus Reading
		                                        
		MesBlock_Temp 				: ARRAY [1..3] OF ARRAY[1..120]  OF WORD; 			// (NA) Temporary Block with multiple modbus reading (Caution : Double Word variables)



	// M_STATEMANAGER//
	
END_VAR

METHOD M_AlarmManagement
//////////////////
// Manages IntelliGen Alarms
/////////////////

VAR 
	// Method local variables (reinitialized at each cycle) 
	FB_AlarmCodeManager : FB_AlarmCodeManager ; 

	KK					: BYTE;		// For Loop 
	
	ComWarning			: BOOL;		// Aggregated Wcommunication warning
	ComAlarm			: BOOL;		// Aggregated communication Alarm

	MesWarningCom: BOOL;
END_VAR

	//Alarm
	
	TON_ComAlarm	(IN:= (AX_ModbusRead[1].ModbusReadAlarm) AND (AX_ModbusRead[2].ModbusReadAlarm) AND (AX_ModbusRead[3].ModbusReadAlarm) , PT:= ParamTempoComAlarm, 	Q=> MesDataExd.MesData.MesAlarmCom) ;	
//	TON_ComWarning	(IN:= (AX_ModbusRead[1].ModbusReadAlarm) OR  (AX_ModbusRead[2].ModbusReadAlarm) OR  (AX_ModbusRead[3].ModbusReadAlarm) , PT:= ParamTempoComWarning, 	Q=>MesWarningCom) ;	

	MesWarningCom :=(AX_ModbusRead[1].ModbusReadAlarm) OR  (AX_ModbusRead[2].ModbusReadAlarm) OR  (AX_ModbusRead[3].ModbusReadAlarm) ; 


	
// ALARM CODE //
	FB_AlarmCodeManager(
		bAlarm1			:= MesDataExd.MesData.MesAlarmImax,  				//  Max I>>0  fault  
		bAlarm2			:= FALSE , 										//
		bAlarm3			:= MesDataExd.MesData.MesAlarmCom , 			// Communication alarm #COM
		bAlarm4			:= MesDataExd.MesData.MesAlarmTCS, 		        // Trip circuit Supervision alarm .     
		bAlarm5			:= FALSE, 										// 
		bAlarm6			:= FALSE, 										// 
		bAlarm7			:= False, 										// 
		bAlarm8			:= False, 										// 
		bAlarm9			:= FALSE, 										//
		bAlarm10		:= FALSE, 										//
		bAlarm11		:= FALSE,                       				//
		bAlarm12		:= FALSE,                       				//
		bAlarm13		:= FALSE, 										//
		bAlarm14		:= FALSE, 										// 
		bAlarm15		:= FALSE , 										// 
		wAlarmCode		=>MesDataExd.MesData.MesAlarmCode);

// WARNING CODE //
	FB_AlarmCodeManager(
 		bAlarm1			:= MesWarningCom,								// Bad communication	#COM			
		bAlarm2			:= FALSE ,										// 
		bAlarm3			:= FALSE , 										//		
		bAlarm4			:= FALSE, 						                //
		bAlarm5			:= FALSE, 						                //
		bAlarm6			:= FALSE, 						                //
		bAlarm7			:= FALSE,                                       //
		bAlarm8			:= FALSE,                                       //
		bAlarm9			:= FALSE,                                       //
		bAlarm10		:= FALSE,                                       //
		bAlarm11		:= FALSE,                                       //
		bAlarm12		:= FALSE,                                       //
		bAlarm13		:= FALSE,                                       //
		bAlarm14		:= FALSE,                                       //
		bAlarm15		:= FALSE,                                       //
		wAlarmCode		=>MesDataExd.MesData.MesWarningCode);	

// EVENT CODE //
	FB_AlarmCodeManager(
 		bAlarm1			:= FALSE,		//				
		bAlarm2			:= FALSE,	    //
		bAlarm3			:= FALSE,		//	
		bAlarm4			:= FALSE, 		//				
		bAlarm5			:= FALSE, 		//				
		bAlarm6			:= FALSE, 		//				
		bAlarm7			:= FALSE,       //
		bAlarm8			:= FALSE,       //
		bAlarm9			:= FALSE,       //
		bAlarm10		:= FALSE,       //
		bAlarm11		:= FALSE,       //
		bAlarm12		:= FALSE,       //
		bAlarm13		:= FALSE,       //
		bAlarm14		:= FALSE,       //
		bAlarm15		:= FALSE,       //
		wAlarmCode		=>MesDataExd.MesData.MesEventCode);
END_METHOD

METHOD M_CP
//////////////////
//  Emulator
/////////////////

VAR 
	// Method local variables (reinitialized at each cycle) 
	
END_VAR


SUPER^.M_CP() ; 




Trig_Cmd_Read(CLK:=IN_CmdToggleRead);
Trig_Cmd_Write(CLK:=IN_CmdToggleWrite);
	
IF Trig_Cmd_Read.Q THEN
	IN_CmdToggleRead := FALSE;
	MesDataExd.MesData.MesCP_Read := NOT MesDataExd.MesData.MesCP_Read;
END_IF


IF Trig_Cmd_Write.Q THEN
	IN_CmdToggleWrite := FALSE;
	MesDataExd.MesData.MesCP_Write := NOT MesDataExd.MesData.MesCP_Write;
END_IF
END_METHOD

METHOD M_Read
//////////////////
//  Read Modbus Variable for PCS . 
/////////////////
VAR 
	// Method local variables (reinitialized at each cycle) 
		
		AX_Addr				: ARRAY[1..3] OF UINT := [138, 		9409, 	171 ];
		AX_Qty				: ARRAY[1..3] OF UINT := [4, 		4, 	36	];
		
	
END_VAR
// CP-Read / Write 



// System BMS 
IF MesDataExd.MesData.MesCP_Read  THEN	

	AX_ModbusRead[1]
	(
		pDestAddr 		:= ADR(MesBlock_Temp[1]),
		sIPAddr 		:= ParamIPAddress,
		tTimeout 		:= ParamTimeout,
		nQuantity 		:= AX_Qty[1],
		ntcpport 		:= ParamTCPPort,
		nMBAddr 		:= AX_Addr[1]-1,
		nUnitID 		:= ParamUnitID,
		cbLength 		:= SIZEOF(MesBlock_Temp[1]),
		ClockRead 		:= ClockRead AND MesDataExd.MesData.MesCP_Read,
		Reset 			:= CmdClearFault_G OR IN_CmdReset_L,
	);
	
	AX_ModbusRead[2]
	(
		pDestAddr 		:= ADR(MesBlock_Temp[2]),
		sIPAddr 		:= ParamIPAddress,
		tTimeout 		:= ParamTimeout,
		nQuantity 		:= AX_Qty[2],
		ntcpport 		:= ParamTCPPort,
		nMBAddr 		:= AX_Addr[2]-1,
		nUnitID 		:= ParamUnitID,
		cbLength 		:= SIZEOF(MesBlock_Temp[2]),
		ClockRead 		:= ClockRead AND MesDataExd.MesData.MesCP_Read,
		Reset 			:= CmdClearFault_G OR IN_CmdReset_L
	);
	
	AX_ModbusRead[3]
	(
		pDestAddr 		:= ADR(MesBlock_Temp[3]),
		sIPAddr 		:= ParamIPAddress,
		tTimeout 		:= ParamTimeout,
		nQuantity 		:= AX_Qty[3],
		ntcpport 		:= ParamTCPPort,
		nMBAddr 		:= AX_Addr[3]-1,
		nUnitID 		:= ParamUnitID,
		cbLength 		:= SIZEOF(MesBlock_Temp[3]),
		ClockRead 		:= ClockRead AND MesDataExd.MesData.MesCP_Read,
		Reset 			:= CmdClearFault_G OR IN_CmdReset_L
	);
	
	
	
		
	
	
	MesDataExd.MesData.MesI1 	:= WORD_TO_REAL(MesBlock_Temp[1][1])/1000*ParamNominalCurrent;
	MesDataExd.MesData.MesI2 	:= WORD_TO_REAL(MesBlock_Temp[1][2])/1000*ParamNominalCurrent;
	MesDataExd.MesData.MesI3 	:= WORD_TO_REAL(MesBlock_Temp[1][3])/1000*ParamNominalCurrent;
	MesDataExd.MesData.MesI0 	:= WORD_TO_REAL(MesBlock_Temp[1][4])/1000*ParamNominalCurrent;
	
	
	MesDataExd.MesData.MesImax1	:= WORD_TO_REAL(MesBlock_Temp[2][1])/1000*ParamNominalCurrent;
	MesDataExd.MesData.MesImax2	:= WORD_TO_REAL(MesBlock_Temp[2][2])/1000*ParamNominalCurrent;
	MesDataExd.MesData.MesImax3	:= WORD_TO_REAL(MesBlock_Temp[2][3])/1000*ParamNominalCurrent;
	MesDataExd.MesData.MesImax0	:= WORD_TO_REAL(MesBlock_Temp[2][4])/1000*ParamNominalCurrent;
	
	
	MesDataExd.MesTransfoAlarm		:= MesBlock_Temp[3][31].0 ;
	MesDataExd.MesSWOpened			:= MesBlock_Temp[3][31].4 ;
	MesDataExd.MesSWClosed			:= MesBlock_Temp[3][31].6 ;
	MesDataExd.MesEarth				:= MesBlock_Temp[3][31].8 ;
	MesDataExd.MesSF6Low			:= MesBlock_Temp[3][31].10;
	MesDataExd.MesSF6Unsufficient	:= MesBlock_Temp[3][31].12;
	MesDataExd.MesTransfoWarning		:= MesBlock_Temp[3][31].14;
	
	MesDataExd.MesClosed	        := MesBlock_Temp[3][30].2;
	MesDataExd.MesOpened	        := MesBlock_Temp[3][30].4;
	MesDataExd.MesComutLocal				:= NOT MesBlock_Temp[3][30].6;
	
	MesDataExd.MesData.MesAlarmImax				:= MesBlock_Temp[3][3].1 ; // Max I ou Max I Inverse. Maintenu jusque l'acquittement.  
	//MesDataExd.MesData.MesAlarmTCS				:=  ; 

END_IF

//MesDataExd.MesData.MesAlarmUminrmUmin	:= ; 

// Properties update
MesDataExd.MesData.MesI := (MesDataExd.MesData.MesI1 + MesDataExd.MesData.MesI2 + MesDataExd.MesData.MesI3)/3 ;
END_METHOD

END_FUNCTION_BLOCK

// ---- 01_Equipement_Library/ProtectRelay/FB_ProtectRelay_SchP3U30.TcPOU
FUNCTION_BLOCK FB_ProtectRelay_SchP3U30 EXTENDS FB_ProtectRelay_Base
//////////////////
// Schneider P30U30 system for High Voltage or Low Voltage Grid Protection. 
//////////////////

VAR_INPUT PERSISTENT
	// Parameters of the Object (instance/model specific) 
	ParamUnitID					: BYTE 		:= 1 ;				(* (NA) Unit ID   							*)	
	ParamTcpPort				: UINT		:= 502;				(* (NA) TCP port 							*)
	ParamIPAddress				: STRING; 						(* (NA)	Config: IP Adress of PV INverter	*)
END_VAR

VAR_OUTPUT
	//Child objects
	OUT_Protect_GTE_LONG_Running: BOOL; 						// Long GTE fault, PP stop for 2m and lost of autorisation 

END_VAR

VAR_INPUT
	// I/O Inputs	
	IN_MesAlarmIMax_IO			: BOOL; 						// I max fault Fault, Losing autorisation and not possible to consumed
	IN_MesAlarmUmin_IO			: BOOL; 						// U min Fault, Keeping autorisation, If we have 3 gte in 30 min ==> Stop fedding and consumed during 2h
	IN_MesAlarmPWH_IO			: BOOL; 						// Defaut wattmétrique
	IN_MesAlarm_IO				: BOOL;							// Equipment alarm
	IN_MesWarning_IO			: BOOL;							// Equipment warning
	
	IN_CmdReset_3GTEFault		: BOOL;							// 3GTE Fault Reset 
		                            			
	MesDataExd		AT %Q* 		: ProtectRelay_SchP30U30; 
	                
END_VAR                         

VAR
	//M_Read		
	FB_ModbusRead	          	: ARRAY[1..3] OF FB_ModbusRead;  // (NA) FB for Modbus Reading
	AX_ModbusReadAlarm			: ARRAY[1..3] OF BOOL;
	AX_ModbusReadAlarmId		: ARRAY[1..3] OF UDINT;		
	
	MesBlock_Temp_1 			: ARRAY [1..120]  OF WORD; 		// (NA) Temporary Block with multiple modbus reading 
	MesBlock_Temp_2 			: ARRAY [1..128] OF WORD; 		// (NA) Temporary Block with multiple modbus reading 
	MesBlock_Temp_3 			: ARRAY [1..128] OF WORD; 		// (NA) Temporary Block with multiple modbus reading 
            			
	//M_EVALUATE                			
	TON_GteIsLong				: TON;
	
	OutErrorMbRead				: ARRAY[1..2] OF BOOL;	
END_VAR

METHOD M_AlarmManagement
//////////////////
// P3U30 Alarms
/////////////////

VAR 
	// Method local variables (reinitialized at each cycle) 
	FB_AlarmCodeManager 	: FB_AlarmCodeManager; 
 	ComWarning				: BOOL;
	ComAlarms				: BOOL;
END_VAR
ComWarning	:= OutErrorMbRead[1] OR OutErrorMbRead[2];
ComAlarms	:= OutErrorMbRead[1];

TON_ComAlarm(IN:= ComAlarms , PT:= ParamTempoComAlarm, Q=>MesDataExd.MesData.MesAlarmCom) ;	

// ALARM CODE //
	FB_AlarmCodeManager(
		bAlarm1				:= FALSE, 								// 
		bAlarm2				:= MesDataExd.MesData.MesAlarmCom,		// Communication alarm #COM
		bAlarm3				:= NOT IN_MesWatchDog_IO,				// WatchDoG TRUE := OK False = Dead #COM
		bAlarm4				:= FALSE,     							// 
		bAlarm5				:= FALSE,         						// 
		bAlarm6				:= FALSE, 								// 
		bAlarm7				:= FALSE, 								// 
		bAlarm8				:= FALSE, 								// 
		bAlarm9				:= FALSE, 								// 
		bAlarm10			:= FALSE, 								// 
		bAlarm11			:= FALSE, 								// 
		bAlarm12			:= FALSE, 								// 
		bAlarm13			:= FALSE, 								// 
		bAlarm14			:= FALSE, 								// 
		bAlarm15			:= FALSE,								//  	
		wAlarmCode			=> MesDataExd.MesData.MesAlarmCode);

// WARNING CODE //
	FB_AlarmCodeManager(
		bAlarm1			:= ComWarning, 								// At least One Register do not responce #COM
		bAlarm2			:= FALSE, 	 								//
		bAlarm3			:= FALSE,									//
		bAlarm4			:= FALSE, 									//
		bAlarm5			:= MesDataExd.MesData.MesAlarmUmin, 		// Min U Fault 
		bAlarm6			:= IN_MesAlarmPWH_IO, 						// Wattmetric fault	
		bAlarm7			:= MesDataExd.MesData.MesAlarmUmin_Long, 	// Long Min U Fault (> 50s)
		bAlarm8			:= FALSE, 									//
		bAlarm9			:= FALSE, 									//
		bAlarm10		:= FALSE, 									//
		bAlarm11		:= FALSE, 									//
		bAlarm12		:= FALSE, 									//
		bAlarm13		:= FALSE, 									//
		bAlarm14		:= FALSE, 									//
		bAlarm15		:= FALSE, 									//
		wAlarmCode		=> MesDataExd.MesData.MesWarningCode);

// EVENT CODE //
	FB_AlarmCodeManager(
		bAlarm1			:=FALSE, 									// 
		bAlarm2			:=FALSE, 									// 
		bAlarm3			:=FALSE, 									// 
		bAlarm4			:=FALSE, 									// 
		bAlarm5			:=FALSE, 									//
		bAlarm6			:=FALSE, 									//
		bAlarm7			:=FALSE, 									//
		bAlarm8			:=FALSE, 									//
		bAlarm9			:=FALSE, 									//
		bAlarm10		:=FALSE, 									//
		bAlarm11		:=FALSE, 									//
		bAlarm12		:=FALSE, 									//
		bAlarm13		:=FALSE, 									//
		bAlarm14		:=FALSE, 									//
		bAlarm15		:=FALSE, 									//
		wAlarmCode		=> MesDataExd.MesData.MesEventCode);
END_METHOD

METHOD M_CP 
VAR_INPUT
END_VAR


SUPER^.M_CP() ; 




Trig_Cmd_Read(CLK:=IN_CmdToggleRead);
Trig_Cmd_Write(CLK:=IN_CmdToggleWrite);
	
IF Trig_Cmd_Read.Q THEN
	IN_CmdToggleRead := FALSE;
	MesDataExd.MesData.MesCP_Read := NOT MesDataExd.MesData.MesCP_Read;
END_IF


IF Trig_Cmd_Write.Q THEN
	IN_CmdToggleWrite := FALSE;
	MesDataExd.MesData.MesCP_Write := NOT MesDataExd.MesData.MesCP_Write;
END_IF
END_METHOD

METHOD M_Evaluate
VAR_INPUT
END_VAR

VAR

END_VAR
// GTE IS LONG AFTER 50S
TON_GteIsLong(IN:=IN_MesAlarmUmin_IO ,PT:=T#50S); 
MesDataExd.MesData.MesAlarmUmin_Long := TON_GteIsLong.Q ; 

//Update MesData
MesDataExd.MesData.MesI			:= (MesDataExd.MesData.MesI1 + MesDataExd.MesData.MesI2 + MesDataExd.MesData.MesI3) / 3 ;
MesDataExd.MesData.MesAlarmUmin := IN_MesAlarmUmin_IO;
MesDataExd.MesData.MesAlarmImax	:= IN_MesAlarmIMax_IO;

MesDataExd.MesPPStop_Lgte 		:= OUT_Protect_GTE_LONG_Running;
END_METHOD

METHOD M_Init
VAR_INPUT
END_VAR
ParamClockReadTime := T#1S;
END_METHOD

METHOD M_Read
//////////////////
//  Method Calls 
/////////////////

VAR 
	MW_Float			: FB_MergeWordsToFloat;
	MW_UInt				: FB_MergeWordsToUint;
	MW_REAL				: FB_MergeWordsToDint;
	
	AX_QTY_MB			: ARRAY[1..4] OF WORD := [120, 3, 7];
	AX_ADR_MB			: ARRAY[1..4] OF WORD := [1990, 4114, 6000]; 	
END_VAR


IF MesDataExd.MesData.MesCP_Read THEN	
	
	FB_ModbusRead[1]
	(
		nTCPPort		:= ParamTcpPort,
		ClockRead		:= MesDataExd.MesData.MesCP_Read AND ClockRead, 
		Reset			:= CmdClearFault_G OR IN_CmdReset_L,
		sIPAddr			:=ParamIPAddress,
		nUnitID			:= 1, 
		tTimeout		:= ParamTimeout,
		nQuantity		:= AX_QTY_MB[1], 
		nMBAddr			:= AX_ADR_MB[1], 
		cbLength		:= SIZEOF(MesBlock_Temp_1), 
		pDestAddr		:= ADR(MesBlock_Temp_1), 
		ModbusReadAlarm	=> AX_ModbusReadAlarm[1], 
		ErrorId			=> AX_ModbusReadAlarmId[1]
	);
	
	FB_ModbusRead[2]
	(
		nTCPPort		:= ParamTcpPort,
		ClockRead		:= MesDataExd.MesData.MesCP_Read AND ClockRead, 
		Reset			:= CmdClearFault_G OR IN_CmdReset_L,
		sIPAddr			:= ParamIPAddress, 
		nUnitID			:= 1, 
		tTimeout		:= ParamTimeout,
		nQuantity		:= AX_QTY_MB[2], 
		nMBAddr			:= AX_ADR_MB[2], 
		cbLength		:= SIZEOF(MesBlock_Temp_2), 
		pDestAddr		:= ADR(MesBlock_Temp_2), 
		ModbusReadAlarm	=>AX_ModbusReadAlarm[2], 
		ErrorId			=> AX_ModbusReadAlarmId[2]
	);
	
	FB_ModbusRead[3]
	(
		nTCPPort		:= ParamTcpPort,
		ClockRead		:= MesDataExd.MesData.MesCP_Read AND ClockRead, 
		Reset			:= CmdClearFault_G OR IN_CmdReset_L,
		sIPAddr			:=ParamIPAddress, 
		nUnitID			:= 1, 
		tTimeout		:= ParamTimeout,
		nQuantity		:= AX_QTY_MB[3], 
		nMBAddr			:= AX_ADR_MB[3], 
		cbLength		:= SIZEOF(MesBlock_Temp_3), 
		pDestAddr		:= ADR(MesBlock_Temp_3), 
		ModbusReadAlarm	=>AX_ModbusReadAlarm[3], 
		ErrorId			=> AX_ModbusReadAlarmId[3]
	);
 
	MesDataExd.MesData.MesWatchdog := WORD_TO_BOOL(MesBlock_Temp_1[11]);
	
	MesDataExd.MesCtoDisparo_Opened     := MesBlock_Temp_1[17].0;
	MesDataExd.MesSpring_Charged	    := MesBlock_Temp_1[17].2;
	MesDataExd.MesInterr_Opened			:= MesBlock_Temp_1[17].3;
//	MesDataExd.MesComutLocal		    := MesBlock_Temp_1[17].5;
	MesDataExd.MesSect_Opened		    := MesBlock_Temp_1[17].6;
	MesDataExd.MesEartch_Opened	        := MesBlock_Temp_1[17].8;
	
	MW_REAL( WORD_STRONG:= MesBlock_Temp_1[19], SIGNED:=FALSE, FIX:=0 , SIZE:=1, VAR_OUT :=MesDataExd.MesData.MesI1);          
	MW_REAL( WORD_STRONG:= MesBlock_Temp_1[20], SIGNED:=FALSE, FIX:=0 , SIZE:=1, VAR_OUT :=MesDataExd.MesData.MesI2);          
	MW_REAL( WORD_STRONG:= MesBlock_Temp_1[21], SIGNED:=FALSE, FIX:=0 , SIZE:=1, VAR_OUT :=MesDataExd.MesData.MesI3);          
	MW_REAL( WORD_STRONG:= MesBlock_Temp_1[22], SIGNED:=FALSE, FIX:=0 , SIZE:=1, VAR_OUT :=MesDataExd.MesData.MesI0);                
	MW_REAL( WORD_STRONG:= MesBlock_Temp_1[24], SIGNED:=FALSE, FIX:=0 , SIZE:=1, VAR_OUT:=MesDataExd.MesData.MesU12);          
	MW_REAL( WORD_STRONG:= MesBlock_Temp_1[25], SIGNED:=FALSE, FIX:=0 , SIZE:=1, VAR_OUT:=MesDataExd.MesData.MesU23);          
	MW_REAL( WORD_STRONG:= MesBlock_Temp_1[26], SIGNED:=FALSE, FIX:=0 , SIZE:=1, VAR_OUT:=MesDataExd.MesData.MesU31);          
	MW_REAL( WORD_STRONG:= MesBlock_Temp_1[27], SIGNED:=FALSE, FIX:=0 , SIZE:=1, VAR_OUT:=MesDataExd.MesV1);                   
	MW_REAL( WORD_STRONG:= MesBlock_Temp_1[28], SIGNED:=FALSE, FIX:=0 , SIZE:=1, VAR_OUT:=MesDataExd.MesV2);                   
	MW_REAL( WORD_STRONG:= MesBlock_Temp_1[29], SIGNED:=FALSE, FIX:=0 , SIZE:=1, VAR_OUT:=MesDataExd.MesV3);                   
	MW_REAL( WORD_STRONG:= MesBlock_Temp_1[30], SIGNED:=FALSE, FIX:=1 , SIZE:=1, VAR_OUT:=MesDataExd.MesV0); 	               
	MW_REAL( WORD_STRONG:= MesBlock_Temp_1[31], SIGNED:=FALSE, FIX:=2 , SIZE:=1, VAR_OUT:=MesDataExd.MesData.MesFreq);                    
	MW_REAL( WORD_STRONG:= MesBlock_Temp_1[32], SIGNED:=TRUE, FIX:=0 , SIZE:=1, VAR_OUT:=MesDataExd.MesP);                     
	MW_REAL( WORD_STRONG:= MesBlock_Temp_1[33], SIGNED:=TRUE, FIX:=0 , SIZE:=1, VAR_OUT:=MesDataExd.MesQ);                     
	MW_REAL( WORD_STRONG:= MesBlock_Temp_1[34], SIGNED:=TRUE, FIX:=0 , SIZE:=1, VAR_OUT:=MesDataExd.MesS);                     
	MW_REAL( WORD_STRONG:= MesBlock_Temp_1[35], SIGNED:=TRUE, FIX:=2 , SIZE:=1, VAR_OUT:=MesDataExd.MesCosPhi);                
	MW_REAL( WORD_STRONG:= MesBlock_Temp_1[36], SIGNED:=FALSE, FIX:=0 , SIZE:=1, VAR_OUT:=MesDataExd.E_P_Prod); 
	MW_REAL( WORD_STRONG:= MesBlock_Temp_1[39], SIGNED:=FALSE, FIX:=0 , SIZE:=1, VAR_OUT:=MesDataExd.E_Q_Prod);               
	MW_REAL( WORD_STRONG:= MesBlock_Temp_1[42], SIGNED:=FALSE, FIX:=0 , SIZE:=1, VAR_OUT:=MesDataExd.E_P_Cons);                               
	MW_REAL( WORD_STRONG:= MesBlock_Temp_1[45], SIGNED:=FALSE, FIX:=0 , SIZE:=1, VAR_OUT:=MesDataExd.E_Q_Cons);
    MW_REAL( WORD_STRONG:= MesBlock_Temp_1[48], SIGNED:=FALSE, FIX:=3 , SIZE:=1, VAR_OUT:=MesDataExd.MesTanPhi);
    MesDataExd.MesComutLocal := WORD_TO_BOOL(MesBlock_Temp_1[58]);  
	
// Maximum values
	MW_REAL( WORD_STRONG:= MesBlock_Temp_2[1], SIGNED:=FALSE, FIX:=0 , SIZE:=1, VAR_OUT :=MesDataExd.MesData.MesImax1);      
	MW_REAL( WORD_STRONG:= MesBlock_Temp_2[2], SIGNED:=FALSE, FIX:=0 , SIZE:=1, VAR_OUT :=MesDataExd.MesData.MesImax2);      
	MW_REAL( WORD_STRONG:= MesBlock_Temp_2[3], SIGNED:=FALSE, FIX:=0 , SIZE:=1, VAR_OUT :=MesDataExd.MesData.MesImax3);
 
// Trip / Alarms
    MesDataExd.MesAlarmImax := MesBlock_Temp_3[1].1; //check
	MesDataExd.MesAlarmImin := MesBlock_Temp_3[1].13;
	MesDataExd.MesAlarmUmax := MesBlock_Temp_3[2].14; //check > >> >>>
	MesDataExd.MesAlarmUmin := MesBlock_Temp_3[3].0; //check < << <<<
	MesDataExd.MesAlarmFmin := MesBlock_Temp_3[4].4; //check < << <<<
	MesDataExd.MesAlarmFmax := MesBlock_Temp_3[4].2; //check < << <<<
	    
// Properties Update 
	MesDataExd.MesU := (MesDataExd.MesData.MesU12 + MesDataExd.MesData.MesU31 + MesDataExd.MesData.MesU23 )/3; 
	MesDataExd.MesData.MesI := (MesDataExd.MesData.MesI1 + MesDataExd.MesData.MesI2 + MesDataExd.MesData.MesI3 )/3; 
	MesDataExd.MesData.MesAlarmImax := MesDataExd.MesAlarmImin OR MesDataExd.MesAlarmImax;
	MesDataExd.MesData.MesAlarmUmin := MesDataExd.MesAlarmUmin OR MesDataExd.MesAlarmUmax OR MesDataExd.MesAlarmFmin OR MesDataExd.MesAlarmFmax;
	
END_IF
END_METHOD

END_FUNCTION_BLOCK

// ---- 01_Equipement_Library/ProtectRelay/FB_ProtectRelay_SepamT20.TcPOU
FUNCTION_BLOCK FB_ProtectRelay_SepamT20 EXTENDS FB_ProtectRelay_Base
//////////////////
// SEPAM system for High Voltage or Low Voltage Grid Protection . 
//////////////////
VAR_INPUT PERSISTENT
	// Parameters of the Object (instance/model specific) 
	 
END_VAR

VAR_OUTPUT
	//Child objects
	OutFBCompleteted						: BOOL;
END_VAR

VAR_INPUT
	InUnitID            : DINT;			// (NA)   ID FOR SEPAM T20 Modbus Unit ID. 
MesDataExd					AT %Q* 		: ProtectRelay_T20;
	
	// I/O Inputs		
END_VAR

VAR
	//M_Read
	FB_ModbusRead_I1						: FB_ReadModbusRTU_V2; 				// (NA) FB for Modbus Reading
	FB_ModbusRead_I2						: FB_ReadModbusRTU_V2; 				// (NA) FB for Modbus Reading
	FB_ModbusRead_I3						: FB_ReadModbusRTU_V2; 				// (NA) FB for Modbus Reading
	ParamTimeoutRTU							: TIME:=T#10S;
	MesBlock1_Temp							: ARRAY [0..36] OF WORD;
	MesBlock2_Temp							: WORD;
	MesBlock3_Temp							: WORD;
	MesModbusAlarmCode						: UDINT;							// (NA) Modbus Read Alarm Code
	MesModbusAlarmCode2						: UDINT;							// (NA) Modbus Read Alarm Code
	MesModbusAlarmCode3						: UDINT;							// (NA) Modbus Read Alarm Code
	ModbusReadAlarm 						: BOOL;								// (NA) Modbus Read Alarm for communications
	ModbusReadAlarm2 						: BOOL;	
	ModbusReadAlarm3 						: BOOL;	
	AX_bRead 								: ARRAY [1..3] OF BOOL;
	CalAllCompleted							: BOOL;
	//M_ALARMMANAGEMENT VARIABLES//

	//M_Execute
	AllNotBusy								: BOOL;
	TP_Read									: TP;
	RTrig									: R_TRIG;
//	ClockRead								: BOOL;
	
	//EValuate//


		
END_VAR

METHOD M_AlarmManagement
//////////////////
// Manages Sepam Alarms. Alarms opens HT CB until Sepam manual Reset . Warning Opens CB-L but does not maintain warning
/////////////////

VAR 
	// Method local variables (reinitialized at each cycle) 
	FB_AlarmCodeManager 	: FB_AlarmCodeManager ; 
 	ComWarning				: BOOL;
	ComAlarms				: BOOL;
END_VAR
ComWarning	:= ModbusReadAlarm OR ModbusReadAlarm2 OR ModbusReadAlarm3;
ComAlarms	:= ModbusReadAlarm OR ModbusReadAlarm2 OR ModbusReadAlarm3;

// ALARM CODE //
	FB_AlarmCodeManager(
		bAlarm1				:= FALSE,									//	
		bAlarm2				:= MesDataExd.MesGlobalWarming > 95 ,		// Calc of Warming TR from Sepam > 95 % OF T° Max				
		bAlarm3				:= ComAlarms ,								// Communication alarm  #COM
		bAlarm4				:= FALSE,     							//
		bAlarm5				:= FALSE,         						// 
		bAlarm6				:= FALSE, 								// 
		bAlarm7				:= FALSE, //
		bAlarm8				:= FALSE, //
		bAlarm9				:= FALSE, //
		bAlarm10			:= FALSE, //
		bAlarm11			:= FALSE, //
		bAlarm12			:= FALSE, //
		bAlarm13			:= FALSE, //
		bAlarm14			:= FALSE, //
		bAlarm15			:= FALSE , 	// 
		wAlarmCode			=>MesDataExd.MesData.MesAlarmCode);

// WARNING CODE //
	FB_AlarmCodeManager(
		bAlarm1			:= ComWarning, 							//  At least One Register do not responce #COM
		bAlarm2			:= FALSE,//  MesDataExd.MesData.MesPartialdefault, 			// Sepam in partial defaut IO, Tor fault
		bAlarm4			:= MesDataExd.MesGlobalWarming > 80, 	// Calc of Warming TR from Sepam > 80 % OF T° Max
		bAlarm5			:= FALSE, //
		bAlarm6			:= FALSE, //
		bAlarm7			:= FALSE, //
		bAlarm8			:= FALSE, //
		bAlarm9			:= FALSE, //
		bAlarm10		:= FALSE, //
		bAlarm11		:= FALSE, //
		bAlarm12		:= FALSE, //
		bAlarm13		:= FALSE, //
		bAlarm14		:= FALSE, //
		bAlarm15		:= FALSE, //
		wAlarmCode		=>MesDataExd.MesData.MesWarningCode);

// EVENT CODE //
	FB_AlarmCodeManager(
		bAlarm1			:=FALSE, 		// 
		bAlarm2			:=FALSE, 		// 
		bAlarm3			:=FALSE, 		// 
		bAlarm4			:=FALSE, 		// 
		bAlarm5			:=FALSE, 
		bAlarm6			:=FALSE, 
		bAlarm7			:=FALSE, 
		bAlarm8			:=FALSE, 
		bAlarm9			:=FALSE, 
		bAlarm10		:=FALSE, 
		bAlarm11		:=FALSE, 
		bAlarm12		:=FALSE, 
		bAlarm13		:=FALSE, 
		bAlarm14		:=FALSE, 
		bAlarm15		:=FALSE, 
		wAlarmCode		=>MesDataExd.MesData.MesEventCode);
END_METHOD

METHOD M_CP 
VAR_INPUT
END_VAR


SUPER^.M_CP() ; 




Trig_Cmd_Read(CLK:=IN_CmdToggleRead);
Trig_Cmd_Write(CLK:=IN_CmdToggleWrite);
	
IF Trig_Cmd_Read.Q THEN
	IN_CmdToggleRead := FALSE;
	MesDataExd.MesData.MesCP_Read := NOT MesDataExd.MesData.MesCP_Read;
END_IF


IF Trig_Cmd_Write.Q THEN
	IN_CmdToggleWrite := FALSE;
	MesDataExd.MesData.MesCP_Write := NOT MesDataExd.MesData.MesCP_Write;
END_IF
END_METHOD

METHOD M_Init
VAR_INPUT
END_VAR
OutFBCompleteted := FALSE;
TP_Read(PT := ParamClockReadTime);
FB_ModbusRead_I1(InTimeout:= ParamTimeoutRTU,
				 InUnitID:= DINT_TO_BYTE(InUnitID),
				 InQuantity:= 36,	
				 InFunctionRead := 1);
				 
FB_ModbusRead_I2(InTimeout:= ParamTimeoutRTU,
				 InUnitID:= DINT_TO_BYTE(InUnitID),
				 InQuantity:= 1,	
				 InFunctionRead := 1);

				 
FB_ModbusRead_I3(InTimeout:= ParamTimeoutRTU,
				 InUnitID:= DINT_TO_BYTE(InUnitID),
				 InQuantity:= 1,	
				 InFunctionRead := 1);
END_METHOD

METHOD M_Read
//////////////////
//  Method Calls 
/////////////////

VAR 
//local variables (reinitialized at each cycle) 
	Busy1 : BOOL;
	Error1: BOOL;
	Busy2 : BOOL;
	Error2: BOOL;
	Busy3 : BOOL;
	Error3: BOOL;
	MW 					: FB_MergeWordsToDint; 
END_VAR
// CP-Read / Write 


IF MesDataExd.MesData.MesCP_Read  THEN	

	AllNotBusy:=TRUE;
	AllNotBusy:=NOT(FB_ModbusRead_I1.OutBusy) AND NOT(FB_ModbusRead_I2.OutBusy) AND NOT(FB_ModbusRead_I3.OutBusy) AND AllNotBusy;
	
	OutFBCompleteted:=FALSE;
	
	// MODBUS REQUEST//
		//First register
			FB_ModbusRead_I1(InClockRead:= ClockRead,				
							InStartAddr:= 16#106,
							InAddrDest := ADR(MesBlock1_Temp),
							OutBusy => Busy1,
							OutErrorMbRead => Error1, 
							OutErrorId => MesModbusAlarmCode
							   );
							
			IF FB_ModbusRead_I1.OutbCompleted THEN
				ModbusReadAlarm := Error1;
				AX_bRead[1] 		:= TRUE;
			ELSIF NOT busy1 AND Error1 THEN
				ModbusReadAlarm := Error1;
			END_IF
		//Seconde Register
			FB_ModbusRead_I2(InClockRead:= ClockRead,				
							InStartAddr:= 16#1004,
							InAddrDest := ADR(MesBlock2_Temp),
							OutBusy => Busy2,
							OutErrorMbRead => Error2, 
							OutErrorId => MesModbusAlarmCode2
							   );		
			IF FB_ModbusRead_I2.OutbCompleted THEN
				ModbusReadAlarm2 := Error2;
				AX_bRead[2] 		:= TRUE;
			ELSIF NOT busy1 AND Error1 THEN
				ModbusReadAlarm2 := Error2;
			END_IF
		
		
		
		//Third Register
			FB_ModbusRead_I3(InClockRead:= ClockRead,				
							InStartAddr:= 16#1007,
							InAddrDest := ADR(MesBlock3_Temp),
							OutBusy => Busy3,
							OutErrorMbRead => Error3, 
							OutErrorId => MesModbusAlarmCode3
							   );		
			IF FB_ModbusRead_I3.OutbCompleted THEN
				ModbusReadAlarm3 := Error3;
				AX_bRead[3] 		:= TRUE;
			ELSIF NOT busy3 AND Error3 THEN
				ModbusReadAlarm3 := Error3;
			END_IF
		
		
	CalAllCompleted :=  AX_bRead[1] AND AX_bRead[2] AND AX_bRead[3];
	OutFBCompleteted := CalAllCompleted;	
	
	//CHECK IF ALL MODBUS REQUESTS ARE FINISHED
		IF (CalAllCompleted) THEN
	//RESETING CLOCK READ FOR EACH REQUEST
			AX_bRead[1]:= FALSE;
			AX_bRead[2]:= FALSE;
			AX_bRead[3]:= FALSE;
			CalAllCompleted := FALSE;
		END_IF
		
	MW( WORD_STRONG:= MesBlock1_Temp[0], SIGNED:=FALSE, FIX:=0 , SIZE:=1, VAR_OUT 	:=MesDataExd.MesData.MesI1);
	MW( WORD_STRONG:= MesBlock1_Temp[1], SIGNED:=FALSE, FIX:=0 , SIZE:=1, VAR_OUT 	:=MesDataExd.MesData.MesI2);
	MW( WORD_STRONG:= MesBlock1_Temp[2], SIGNED:=FALSE, FIX:=0 , SIZE:=1, VAR_OUT 	:=MesDataExd.MesData.MesI3);
	MW( WORD_STRONG:= MesBlock1_Temp[33], SIGNED:=FALSE, FIX:=2 , SIZE:=1, VAR_OUT	:=MesDataExd.MesData.MesFreq);
	MW( WORD_STRONG:= MesBlock1_Temp[34], SIGNED:=TRUE, FIX:=0 , SIZE:=1, VAR_OUT 	:=MesDataExd.MesP);
	MW( WORD_STRONG:= MesBlock1_Temp[35], SIGNED:=TRUE, FIX:=0 , SIZE:=1, VAR_OUT 	:=MesDataExd.MesQ);
	MW( WORD_STRONG:= MesBlock1_Temp[36], SIGNED:=TRUE, FIX:=0 , SIZE:=1, VAR_OUT 	:=MesDataExd.MesS);
	MW( WORD_STRONG:= MesBlock2_Temp, SIGNED:=FALSE, FIX:=-1 , SIZE:=1, VAR_OUT 	:=MesDataExd.MesTripProtec);
	MW( WORD_STRONG:= MesBlock3_Temp, SIGNED:=FALSE, FIX:=0 , SIZE:=1, VAR_OUT 		:=MesDataExd.MesGlobalWarming);

END_IF
END_METHOD

END_FUNCTION_BLOCK

// ---- 01_Equipement_Library/ProtectRelay/FB_ProtectRelay_Siprotec.TcPOU
FUNCTION_BLOCK FB_ProtectRelay_Siprotec EXTENDS FB_ProtectRelay_Base
// Hypothèse : défaut GTE entraîne ouverture automatique CB

VAR_INPUT PERSISTENT
	ParamTimeGteIsLong					: TIME := T#60S; 	(* Time after which a GTE fault is considered long *)
	ParamTimeBeforeReconnect			: TIME := T#5M;		(* Time after a Short GTE when we can reconnect *)
	                                                                                                        
	// Parameters of the Object (instance specific)                                                         
	ParamIPAddress			: STRING := '127.0.0.1'; 		(* (NA)Config: IP Adress of RPN                 *)
	ParamnTcpPort			: UINT := 502;					(* TCP Port                                     *)
	ParamUnitID 			: BYTE  := 1; 			  		(* (NA)   SMA Modbus Unit ID.                   *)
	ParamInvNum				: BYTE ; 						(* (NA) Config :Numerous of the ESS in the HPP  *)
	ParamOffsetRegisters	: UINT;
	ParamCommunicating		: BOOL;
	ParamAlarmUmin_NC		: BOOL;
	ParamAlarmImax_NC		: BOOL;
	ParamWatchdog_NC		: BOOL;
	
END_VAR


VAR_INPUT
	IN_MesAlarmIMax_IO						: BOOL; // C 13 100 Fault (internal)
	IN_MesAlarmUmin_IO						: BOOL; // GTE Fault (external)
	IN_MesComut_IO							: BOOL;
	IN_TCSAlarm								: BOOL; // Alarme TCS (Supervision circuit de déclenchement)
	IN_VrAnomaly							: BOOL; // Anomalie VR (Tension résiduelle)
	IN_TripSynthesis						: BOOL; // Trip Synthesis
	IN_CmdReset_3GTEFault					: BOOL; // 3GTE Fault Reset 
	
	MesDataExd						: ProtectRelay_Siprotec;
END_VAR                         		
VAR_OUTPUT                      		
	OUT_CmdCloseMainCB						: BOOL;	// Cmd to close the main CB : if after 60s Gte is short OR if gte long AND after the grid stab
	OUT_CmdOpenMainCB						: BOOL;
	OUT_CmdAutoRecouplage_GteShort			: BOOL;	// 
	OUT_MesC13100Fault_IO					: BOOL;
END_VAR                         		
VAR 
	// M_READ VARIABLES 

		FB_ModbusRead_RPN_3X		: FB_ModbusReadInputRegs ; 	// (NA) FB for Modbus Reading
		
		MesBlock_Temp 				: ARRAY[1..4] OF ARRAY [1..125] OF WORD ; 			// (NA) Temporary Block with multiple modbus reading (Caution : Double Word variables)
		
		AX_Error					: ARRAY[1..4] OF BOOL;
		AX_ErrorID					: ARRAY[1..4] OF UDINT;
                            		
	//EVALUATE VARIABLES        	
		TON_Communication_Alarm			: TON;
		// GTE                  		
		
	//M_EVALUATE                			
		TON_GteIsLong							: TON;
		
		FB_3GTE							: FB_CountNinTimeWindow; 
		
			

		MesFreq_Old						: REAL;
END_VAR

METHOD M_AlarmManagement
//////////////////
// Manages Sepam Alarms. Alarms opens HT CB until Sepam manual Reset . Warning Opens CB-L but does not maintain warning
/////////////////

VAR 
	// Method local variables (reinitialized at each cycle) 
	FB_AlarmCodeManager 	: FB_AlarmCodeManager ; 

 
END_VAR
IF ParamCommunicating THEN
	TON_Communication_Alarm(in:=MesFreq_Old = MesDataExd.MesFreq, PT := T#3S, Q=> MesDataExd.MesData.MesAlarmCom);
	IF MesFreq_Old <> MesDataExd.MesFreq THEN
		MesFreq_Old := MesDataExd.MesFreq;
	END_IF
ELSE
	MesDataExd.MesData.MesAlarmCom := FALSE;

END_IF


MesDataExd.MesComutLocal			:= IN_MesComut_IO ; 
MesDataExd.MesTCSAlarm				:= IN_TCSAlarm;
MesDataExd.MesVrAnomaly				:= IN_VrAnomaly;
MesDataExd.MesTripSynthesis			:= IN_TripSynthesis;

// ALARM CODE //
	FB_AlarmCodeManager(
		bAlarm1			:=MesdataExd.MesData.MesAlarmUmin, 		// GTE Fault in Siprotec
		bAlarm2			:=MesDataExd.MesData.MesAlarmUmin_Long, 	// GTE Fault Long
		bAlarm3			:=FALSE,
		bAlarm4			:=MesDataExd.MesData.MesAlarmImax, 	// C13100 Fault in Siprotec
		bAlarm5			:=MesDataExd.MesData.MesWatchdog,	// Watchdog fault if FALSE
		bAlarm6			:=MesDataExd.MesData.MesAlarmCom,	// Communication alarm: no comm at all for 3s
		bAlarm7			:=MesDataExd.MesTCSAlarm,           // Alarme TCS (Supervision circuit de déclenchement)
		bAlarm8			:=MesDataExd.MesVrAnomaly,      	// Anomalie VR (tension résiduelle)
		bAlarm9			:=MesDataExd.MesTripSynthesis,      // Trip Synthesis
		bAlarm10		:=FALSE,                        	//
		bAlarm11		:=FALSE,                        	//
		bAlarm12		:=FALSE,                        	//
		bAlarm13		:=FALSE,                        	//
		bAlarm14		:=FALSE,                        	//
		bAlarm15		:=FALSE, 							//
		wAlarmCode		=> MesDataExd.MesData.MesAlarmCode);

// WARNING CODE //
	FB_AlarmCodeManager(		
		bAlarm1			:=MesDataExd.MesComutLocal, 	// COMMUTATOR IN LOCAL
		bAlarm2			:=FALSE,						//
		bAlarm3			:=FALSE,                        //
		bAlarm4			:=FALSE,                        //
		bAlarm5			:=FALSE,                        //
		bAlarm6			:=FALSE,                        //
		bAlarm7			:=FALSE,                        //
		bAlarm8			:=FALSE,                        //
		bAlarm9			:=FALSE,                        //
		bAlarm10		:=FALSE,                        //
		bAlarm11		:=FALSE,                        //
		bAlarm12		:=FALSE,                        //
		bAlarm13		:=FALSE,                        //
		bAlarm14		:=FALSE,                        //
		bAlarm15		:=FALSE,                        //
		wAlarmCode		=> MesDataExd.MesData.MesWarningCode);
END_METHOD

METHOD M_CP 
VAR_INPUT
END_VAR


SUPER^.M_CP() ; 




Trig_Cmd_Read(CLK:=IN_CmdToggleRead);
Trig_Cmd_Write(CLK:=IN_CmdToggleWrite);
	
IF Trig_Cmd_Read.Q THEN
	IN_CmdToggleRead := FALSE;
	MesDataExd.MesData.MesCP_Read := NOT MesDataExd.MesData.MesCP_Read;
END_IF


IF Trig_Cmd_Write.Q THEN
	IN_CmdToggleWrite := FALSE;
	MesDataExd.MesData.MesCP_Write := NOT MesDataExd.MesData.MesCP_Write;
END_IF
END_METHOD

METHOD M_Evaluate
VAR_INPUT
END_VAR
VAR
	MesOneFault 			: BOOL;		// at least one fault active;
	PDLState				: BYTE;		//  Bit0: Decouplée , Bit1: Couplée ,BIT2 : effacée
	KK: INT;
	btest : bool;
END_VAR

// GTE IS LONG AFTER 50S
TON_GteIsLong(IN:=IN_MesAlarmUmin_IO ,PT:=T#50S); 
MesDataExd.MesData.MesAlarmUmin_Long := TON_GteIsLong.Q ; 

FB_3GTE(IN_bInput := IN_MesAlarmUmin_IO , IN_bReset := IN_CmdReset_3GTEFault , IN_CountMax := 3 , ParamTimeToMeasure := T#30M , OUT_FlagNinT =>MesDataExd.MesData.MesAlarm_GTE3Time ) ; 
	
//Update MesData
MesDataExd.MesI			:= (MesDataExd.MesI1 + MesDataExd.MesI2 + MesDataExd.MesI3) / 3 ;

	IF ParamAlarmUmin_NC THEN
		MesDataExd.MesData.MesAlarmUmin	:= NOT IN_MesAlarmUmin_IO ; 
	ELSE
		MesDataExd.MesData.MesAlarmUmin	:= IN_MesAlarmUmin_IO ; 
	END_IF
	
	IF ParamAlarmImax_NC THEN
		MesDataExd.MesData.MesAlarmImax	:= NOT IN_MesAlarmIMax_IO ; 
	ELSE
		MesDataExd.MesData.MesAlarmImax	:= IN_MesAlarmIMax_IO ; 
	END_IF
	
	IF ParamWatchdog_NC THEN
		MesDataExd.MesData.MesWatchdog	:= NOT IN_MesWatchDog_IO ; 
	ELSE
		MesDataExd.MesData.MesWatchdog	:= IN_MesWatchDog_IO ; 
	END_IF
END_METHOD

METHOD M_Execute
//////////////////
//  Method Calls 
/////////////////

VAR 
	// Method local variables (reinitialized at each cycle) 

END_VAR
SUPER^.M_Execute() ;
END_METHOD

METHOD M_Init
VAR_INPUT
END_VAR

VAR
	KK: INT;
END_VAR
//A1_ProtectRelay.ParamClockReadTime := T#2S ; 
//A1_ProtectRelay.ParamTimeOut	:= T#5S ; 
//A1_ProtectRelay.ParamUnitID := 1 ; 
//A1_ProtectRelay.ParamAlarmUmin_NC:= TRUE;
//A1_ProtectRelay.ParamAlarmImax_NC:= TRUE;
//A1_ProtectRelay.ParamWatchdog_NC:= TRUE;
END_METHOD

METHOD M_Read
//////////////////
//  Method Calls 
/////////////////

VAR 
	// Method local variables (reinitialized at each cycle)
	i 					: INT;
	MW					: FB_MergeWordsToDint; 
	AX_Adr				: ARRAY[1..4] OF WORD 		:= [32,	00001,	00000,	00129];
	AX_Qty				: ARRAY[1..4] OF WORD		:= [1,		107,	16,		83];
END_VAR
// MODBUS REQUESTS//
IF MesDataExd.MesData.MesCP_Read THEN
		
	FB_ModbusRead_RPN_3X(
		nTcpPort 		:= ParamnTcpPort,
		tTimeout		:= ParamTimeout,
		nUnitID			:= ParamUnitID, 
		sIPAddr			:= ParamIPAddress , 
		ClockRead		:= ClockRead AND MesDataExd.MesData.MesCP_Read,
		Reset			:= CmdClearFault_G ,
		nQuantity		:= AX_Qty[3], 
		nMBAddr			:= AX_Adr[3] + ParamOffsetRegisters,  
		cbLength		:= SIZEOF(MesBlock_Temp[3]) , 
		pDestAddr		:= ADR(MesBlock_Temp[3]) , 
		ModbusReadAlarm	=> AX_Error[3] , 
		ErrorId			=> AX_ErrorID[3]
	);
			
	// MODBUS BLOCKS SEPARATION	
		
		MW(WORD_STRONG := MesBlock_Temp[3][1], FIX := 1, SIGNED := TRUE, VAR_OUT := MesdataExd.MesI1);
		MW(WORD_STRONG := MesBlock_Temp[3][2], FIX := 1, SIGNED := TRUE, VAR_OUT := MesdataExd.MesI2);
		MW(WORD_STRONG := MesBlock_Temp[3][3], FIX := 1, SIGNED := TRUE, VAR_OUT := MesdataExd.MesI3);
		MW(WORD_STRONG := MesBlock_Temp[3][4], FIX := 1, SIGNED := TRUE, VAR_OUT := MesdataExd.MesIn);
		MW(WORD_STRONG := MesBlock_Temp[3][5], FIX := 2, SIGNED := TRUE, VAR_OUT := MesdataExd.MesV1);
		MW(WORD_STRONG := MesBlock_Temp[3][6], FIX := 2, SIGNED := TRUE, VAR_OUT := MesdataExd.MesV2);
		MW(WORD_STRONG := MesBlock_Temp[3][7], FIX := 2, SIGNED := TRUE, VAR_OUT := MesdataExd.MesV3);
		MW(WORD_STRONG := MesBlock_Temp[3][8], FIX := 2, SIGNED := TRUE, VAR_OUT := MesdataExd.MesU12);
		MW(WORD_STRONG := MesBlock_Temp[3][9], FIX := 2, SIGNED := TRUE, VAR_OUT := MesdataExd.MesU23);
		MW(WORD_STRONG := MesBlock_Temp[3][10], FIX := 2, SIGNED := TRUE, VAR_OUT := MesdataExd.MesU31);
		MW(WORD_STRONG := MesBlock_Temp[3][11], FIX := 2, SIGNED := TRUE, VAR_OUT := MesdataExd.MesUn);
	//	MW(WORD_STRONG := MesBlock_Temp[3][12], FIX := -1, SIGNED := TRUE, VAR_OUT := MesdataExd.MesP);
		MW(WORD_STRONG := MesBlock_Temp[3][13], FIX := -1, SIGNED := TRUE, VAR_OUT := MesdataExd.MesQ);
		MW(WORD_STRONG := MesBlock_Temp[3][14], FIX := -1, SIGNED := TRUE, VAR_OUT := MesdataExd.MesS);
		MW(WORD_STRONG := MesBlock_Temp[3][15], FIX := 2, SIGNED := TRUE, VAR_OUT := MesdataExd.MesFreq);
		MW(WORD_STRONG := MesBlock_Temp[3][16], FIX := 4, SIGNED := TRUE, VAR_OUT := MesdataExd.MesCosPhi);
		
	IF abs(MesDataExd.MesCosPhi) < 1 THEN
		MesdataExd.MesP := (MesDataExd.MesI1*MesDataExd.MesV1 + MesDataExd.MesI2*MesDataExd.MesV2 + MesDataExd.MesI3*MesDataExd.MesV3 )* abs(MesDataExd.MesCosPhi);
	ELSE
		MesdataExd.MesP := (MesDataExd.MesI1*MesDataExd.MesV1 + MesDataExd.MesI2*MesDataExd.MesV2 + MesDataExd.MesI3*MesDataExd.MesV3 );
	END_IF
		

END_IF
END_METHOD

END_FUNCTION_BLOCK

// ---- 01_Equipement_Library/ProtectRelay/FB_ProtectRelay_SMNS7SL86.TcPOU
FUNCTION_BLOCK FB_ProtectRelay_SMNS7SL86 EXTENDS FB_ProtectRelay_Base
//////////////////
// Siemens 7SJ82 protection relay
//////////////////

VAR_INPUT PERSISTENT
	// Parameters of the Object (instance/model specific) 
	{attribute 'OPC.UA.DA' := '1'} 
	ParamTcpPort					: UINT		:= 502;				(* (NA) TCP port*)
	{attribute 'OPC.UA.DA' := '1'} 
	ParamIPAddress					: STRING; 						(* (NA)Config: IP Adress of PV INverter	*)
	{attribute 'OPC.UA.DA' := '1'} 
	ParamUnitID 					: BYTE; 						(* (NA) Modbus Unit ID *)
	ParamNumInv						: BYTE;             			(* (NA) Number of inverters*)
END_VAR

VAR_OUTPUT
	//Child objects
	OUT_Protect_GTE_LONG_Running			: BOOL; 							// Long GTE fault, PP stop for 2m and lost of autorisation 
END_VAR

VAR_INPUT
	// I/O Inputs	
	IN_MesAlarmIMax_IO						: BOOL; 							// I max fault Fault, Losing autorisation and not possible to consumed
	IN_MesAlarmUmin_IO						: BOOL; 							// U min Fault, Keeping autorisation, If we have 3 gte in 30 min ==> Stop fedding and consumed during 2h
	IN_MesAlarmPWH_IO						: BOOL; 							// Defaut wattmétrique
	                                                								                                                	
	IN_CmdReset_3GTEFault					: BOOL; 							// 3GTE Fault Reset 
	
	MesDataExd				AT %Q* 			: ProtectRelay_SMNS7L86;	
	IN_MesAlarm_IO							: BOOL;
	IN_MesWarning_IO						: BOOL;
END_VAR

VAR
	//M_Read
	Trig_Read								: R_TRIG;

    ModbusRead_RPN_1X						: ARRAY[1..1] OF FB_ModbusReadCoils ;  
	AX_ADR_1X								: ARRAY[1..1] OF WORD := [110];				// (NA) Quantity of blocks to read
	AX_QTY_1X								: ARRAY[1..1] OF WORD := [18];				// (NA) Quantity of blocks to read
	BlockModbus_RPN_1X						: ARRAY[1..1] OF ARRAY[1..120] OF WORD;
	Error_1X								: ARRAY[1..1] OF BOOL;
	ErrorID_1X								: ARRAY[1..1] OF BOOL;

	
    ModbusRead_RPN_3X						: ARRAY[1..1] OF FB_ModbusRead ;  
	AX_ADR_3X								: ARRAY[1..1] OF WORD := [2025];				// (NA) Quantity of blocks to read
	AX_QTY_3X								: ARRAY[1..1] OF WORD := [22];				// (NA) Quantity of blocks to read
	BlockModbus_RPN_3X						: ARRAY[1..1] OF ARRAY[1..120] OF WORD;
	Error_3X								: ARRAY[1..1] OF BOOL;
	ErrorID_3X								: ARRAY[1..1] OF BOOL;
                               			
	                            			
	AX_Error								: ARRAY[1..4] OF BOOL;
	AX_ErrorID								: ARRAY[1..4] OF UDINT;
           
END_VAR

METHOD M_AlarmManagement
//////////////////
// Managing alarms in this method. 
//////////////////

VAR 
	// Method local variables (reinitialized at each cycle) 
	FB_AlarmCodeManager 	: FB_AlarmCodeManager; 

	bComAlarm: BOOL;
	bComWarning: BOOL;
END_VAR
bComAlarm := Error_1X[1] AND Error_3X[1];
bComWarning := Error_1X[1] OR Error_3X[1];

TON_ComAlarm(IN := bComAlarm, PT := T#30S, Q=> MesDataExd.MesData.MesAlarmCom);
TON_ComWarning(IN := bComWarning, PT := T#30S, Q=> MesDataExd.MesData.MesWarningCom);

// ALARM CODE //
	FB_AlarmCodeManager(
		bAlarm1				:= MesDataExd.MesAlarmTripCircuit1,									// Trip circuit 1 Fail
		bAlarm2				:= MesDataExd.MesAlarmTripCircuit2,									// Trip circuit 2 Fail
		bAlarm3				:= MesDataExd.MesTrip_ANSI_5051,									// ANSI 50/51 Trip
		bAlarm4				:= MesDataExd.MesTrip_ANSI_87L,     								// ANSI 87L Trip
		bAlarm5				:= MesDataExd.MesTrip_ANSI_59,         								// ANSI 59 Trip
		bAlarm6				:= MesDataExd.MesTrip_ANSI_59n, 									// ANSI 59N Trip
		bAlarm7				:= MesDataExd.MesTrip_ANSI_81U, 									// ANSI 81U Trip
		bAlarm8				:= MesDataExd.MesTrip_ANSI_81O, 									// ANSI 81O Trip
		bAlarm9				:= MesDataExd.MesData.MesAlarmCom, 									// Communication Alarm
		bAlarm10			:= FALSE, 									//    
		bAlarm11			:= FALSE, 									//                
		bAlarm12			:= FALSE, 									// 
		bAlarm13			:= FALSE, 									// 
		bAlarm14			:= FALSE, 									// 
		bAlarm15			:= FALSE,									// 
		wAlarmCode			=>MesDataExd.MesData.MesAlarmCode);                                                      
                                                                           
// WARNING CODE //                                                         
	FB_AlarmCodeManager(                                                   
		bAlarm1			:= MesDataExd.MesData.MesWarningCom,	 									// Communication Warning
		bAlarm2			:= FALSE,										// 
		bAlarm4			:= FALSE, 										//
		bAlarm5			:= FALSE, 										//
		bAlarm6			:= FALSE,			 							// 	
		bAlarm7			:= FALSE, 										// 
		bAlarm8			:= FALSE, 										// 
		bAlarm9			:= FALSE, 										//
		bAlarm10		:= FALSE, 										//
		bAlarm11		:= FALSE, 										//
		bAlarm12		:= FALSE, 										//
		bAlarm13		:= FALSE, 										//
		bAlarm14		:= FALSE, 										//
		bAlarm15		:= FALSE, 										//
		wAlarmCode		=>MesDataExd.MesData.MesWarningCode);

// EVENT CODE //
	FB_AlarmCodeManager(
		bAlarm1			:=MesDataExd.MesOpened_52, 										// CB Opened							
		bAlarm2			:=MesDataExd.MesClosed_52, 										// CB Closed                			
		bAlarm3			:=MesDataExd.MesOpened_89, 										// Disconnecting switch opened       
		bAlarm4			:=MesDataExd.MesClosed_89, 										// Disconnecting switch closed       
		bAlarm5			:=MesDataExd.MesOpened_89T, 									// Earthing switch Opened            
		bAlarm6			:=MesDataExd.MesClosed_89T, 									// Earthing switch Closed            
		bAlarm7			:=MesDataExd.MesLocalMode, 										// Local mode              			
		bAlarm8			:=MesDataExd.MesSpring_Loaded, 									// Spring charged                    
		bAlarm9			:=FALSE, 										//
		bAlarm10		:=FALSE, 										//
		bAlarm11		:=FALSE, 										//
		bAlarm12		:=FALSE, 										//
		bAlarm13		:=FALSE, 										//
		bAlarm14		:=FALSE, 										//
		bAlarm15		:=FALSE, 										//
		wAlarmCode		=>MesDataExd.MesData.MesEventCode);
END_METHOD

METHOD M_CP 
VAR_INPUT
END_VAR


SUPER^.M_CP() ; 




Trig_Cmd_Read(CLK:=IN_CmdToggleRead);
Trig_Cmd_Write(CLK:=IN_CmdToggleWrite);
	
IF Trig_Cmd_Read.Q THEN
	IN_CmdToggleRead := FALSE;
	MesDataExd.MesData.MesCP_Read := NOT MesDataExd.MesData.MesCP_Read;
END_IF


IF Trig_Cmd_Write.Q THEN
	IN_CmdToggleWrite := FALSE;
	MesDataExd.MesData.MesCP_Write := NOT MesDataExd.MesData.MesCP_Write;
END_IF
END_METHOD

METHOD M_Evaluate
VAR_INPUT
END_VAR

//Update MesData
MesDataExd.MesData.MesI			:= (MesDataExd.MesData.MesI1 + MesDataExd.MesData.MesI2 + MesDataExd.MesData.MesI3) / 3 ;
MesDataExd.MesData.MesTripped 	:= MesDataExd.MesData.MesAlarmImax OR  MesDataExd.MesData.MesAlarmUmin OR  MesDataExd.MesData.MesAlarmCode.6;
END_METHOD

METHOD M_Init
VAR_INPUT
END_VAR
END_METHOD

METHOD M_Read
//////////////////
//  Read Method 
/////////////////

VAR 
	I 					: INT;
	MW					: FB_MergeWordsToFloat; 
	
	bAlarm				: BOOL;

END_VAR

// MODBUS REQUESTS//
IF MesDataExd.MesData.MesCP_Read THEN
		// The read of the equipment's measurements is done in the gateway
	ModbusRead_RPN_1X[1](
		pDestAddr 	:= ADR(BlockModbus_RPN_1X[1]),
		cbLength	:= SIZEOF(BlockModbus_RPN_1X[1]),
		sIPAddr		:= ParamIPAddress,
		tTimeout 	:= ParamTimeOut,
		nTcpPort 	:= ParamTcpPort,
		nQuantity 	:= AX_QTY_1X[1],
		nMBAddr		:= AX_ADR_1X[1],
		nUnitID		:= ParamUnitID,
		ClockRead	:= ClockRead,
		ModbusReadAlarm => Error_1X[1]
		
	);
	
	
	ModbusRead_RPN_3X[1](
		pDestAddr 	:= ADR(BlockModbus_RPN_3X[1]),
		cbLength	:= SIZEOF(BlockModbus_RPN_3X[1]),
		sIPAddr		:= ParamIPAddress,
		tTimeout 	:= ParamTimeOut,
		nTcpPort 	:= ParamTcpPort,
		nQuantity 	:= AX_QTY_3X[1],
		nMBAddr		:= AX_ADR_3X[1],
		nUnitID		:= ParamUnitID,
		ClockRead	:= ClockRead,
		ModbusReadAlarm => Error_3X[1]
	);
	
	// MODBUS BLOCKS SEPARATION	
		
	MesDataExd.MesOpened_52					:= BlockModbus_RPN_1X[1][1].0;			(*CB Opened							*)            
	MesDataExd.MesClosed_52					:= BlockModbus_RPN_1X[1][1].1;          (*CB Closed                			*)
	MesDataExd.MesOpened_89					:= BlockModbus_RPN_1X[1][1].2;		    (*Disconnecting switch opened       *)
	MesDataExd.MesClosed_89 				:= BlockModbus_RPN_1X[1][1].3;		    (*Disconnecting switch closed       *)
    MesDataExd.MesOpened_89T				:= BlockModbus_RPN_1X[1][1].4;          (*Earthing switch Opened            *)
    MesDataExd.MesClosed_89T				:= BlockModbus_RPN_1X[1][1].5;          (*Earthing switch Closed            *)
    MesDataExd.MesLocalMode		    		:= BlockModbus_RPN_1X[1][1].6;          (*Local mode              			*)
    MesDataExd.MesSpring_Loaded				:= BlockModbus_RPN_1X[1][1].7;          (*Spring charged                    *)
    MesDataExd.MesAlarmTripCircuit1			:= BlockModbus_RPN_1X[1][1].8;          (*Trip circuit 1 Fail              	*)
    MesDataExd.MesAlarmTripCircuit2			:= BlockModbus_RPN_1X[1][1].9;          (*Trip circuit 2 Fail               *)
	MesDataExd.MesTrip_ANSI_5051			:= BlockModbus_RPN_1X[1][1].10;         (*ANSI 50/51 Trip                   *)
	MesDataExd.MesTrip_ANSI_87L				:= BlockModbus_RPN_1X[1][1].11;         (*ANSI 87L Trip                     *)
	MesDataExd.MesTrip_ANSI_59				:= BlockModbus_RPN_1X[1][1].12;         (*ANSI 59 Trip                      *)
	MesDataExd.MesTrip_ANSI_59n				:= BlockModbus_RPN_1X[1][1].13;         (*ANSI 59N Trip                     *)
	MesDataExd.MesTrip_ANSI_81U				:= BlockModbus_RPN_1X[1][1].14;         (*ANSI 81U Trip                     *)
	MesDataExd.MesTrip_ANSI_81O				:= BlockModbus_RPN_1X[1][1].15;         (*ANSI 81O Trip                     *)
	MesDataExd.MesTrip_ANSI_27				:= BlockModbus_RPN_1X[1][2].1;         (*ANSI 27 Trip                     *)
	                                                                                
	
	
	MW(WORD_STRONG := BlockModbus_RPN_3X[1][  1], WORD_WEAK := BlockModbus_RPN_3X[1][  2], var_out := MesDataExd.MesData.MesI1);
	MW(WORD_STRONG := BlockModbus_RPN_3X[1][  3], WORD_WEAK := BlockModbus_RPN_3X[1][  4], var_out := MesDataExd.MesData.MesI2);		
	MW(WORD_STRONG := BlockModbus_RPN_3X[1][  5], WORD_WEAK := BlockModbus_RPN_3X[1][  6], var_out := MesDataExd.MesData.MesI3);	
	MW(WORD_STRONG := BlockModbus_RPN_3X[1][  7], WORD_WEAK := BlockModbus_RPN_3X[1][  8], var_out := MesDataExd.MesV1);
	MW(WORD_STRONG := BlockModbus_RPN_3X[1][  9], WORD_WEAK := BlockModbus_RPN_3X[1][ 10], var_out := MesDataExd.MesV2);		
	MW(WORD_STRONG := BlockModbus_RPN_3X[1][ 11], WORD_WEAK := BlockModbus_RPN_3X[1][ 12], var_out := MesDataExd.MesV3);		
	MW(WORD_STRONG := BlockModbus_RPN_3X[1][ 13], WORD_WEAK := BlockModbus_RPN_3X[1][ 14], var_out := MesDataExd.MesP);		
	MW(WORD_STRONG := BlockModbus_RPN_3X[1][ 15], WORD_WEAK := BlockModbus_RPN_3X[1][ 16], var_out := MesDataExd.MesQ);		
	MW(WORD_STRONG := BlockModbus_RPN_3X[1][ 17], WORD_WEAK := BlockModbus_RPN_3X[1][ 18], var_out := MesDataExd.MesS);	
	MW(WORD_STRONG := BlockModbus_RPN_3X[1][ 19], WORD_WEAK := BlockModbus_RPN_3X[1][ 20], var_out := MesDataExd.MesCosPhi);	
	MW(WORD_STRONG := BlockModbus_RPN_3X[1][ 21], WORD_WEAK := BlockModbus_RPN_3X[1][ 22], var_out := MesDataExd.MesData.MesFreq);	

END_IF

MesDataExd.MesP := - MesDataExd.MesP *1000;
MesDataExd.MesQ := - MesDataExd.MesQ *1000;
END_METHOD

END_FUNCTION_BLOCK

// ---- 01_Equipement_Library/ProtectRelay/FB_ProtectRelay_VIP410.TcPOU
FUNCTION_BLOCK FB_ProtectRelay_VIP410 EXTENDS FB_ProtectRelay_Base
//////////////////
// SEPAM system for High Voltage or Low Voltage Grid Protection . 
//////////////////
VAR_INPUT PERSISTENT
	{attribute 'OPC.UA.DA' := '1'} 
	ParamTcpPort				: UINT:=502;		(* (NA) Tcp port *)
	{attribute 'OPC.UA.DA' := '1'} 
	ParamIPAddress				: STRING;       	(* (NA) IP address*)
	{attribute 'OPC.UA.DA' := '1'} 
	ParamUnitID					: BYTE;         	(* (NA) Unit ID*)
	{attribute 'OPC.UA.DA' := '1'}
	ParamClockInputTime 		: TIME:= TIME#5S;   (* (Time) Read Modbus Frequency*)
END_VAR

VAR_OUTPUT
	
END_VAR

VAR_INPUT
	
	MesDataExd		AT %Q* 		: ProtectRelay_VIP410;

	IN_MesTrip_IO				: BOOL ; 
END_VAR

VAR
	

	FB_ModbusRead	          	: ARRAY[1..4] OF FB_ModbusRead; 
	ClockReadInput				: BOOL;

	MesBlock1_Temp 				: ARRAY [1..1] OF WORD ; 
	MesBlock2_Temp 				: ARRAY [1..20] OF WORD ; 
	MesBlock3_Temp 				: ARRAY [1..8] OF WORD ; 
	MesBlock4_Temp 				: ARRAY [1..2] OF WORD ; 
	AX_ModbusReadAlarm			: ARRAY[1..4] OF BOOL;
	AX_ModbusReadAlarmId		: ARRAY[1..4] OF UDINT;	
END_VAR

METHOD M_AlarmManagement
//////////////////
// Manages Sepam Alarms. Alarms opens HT CB until Sepam manual Reset . Warning Opens CB-L but does not maintain warning
/////////////////

